DATA_BLOCK "MEStoPLC"
{ S7_Optimized_Access := 'FALSE' }
VERSION : 0.1
NON_RETAIN
   STRUCT 
      "MES.Load_Station1PartOK" : Bool;
      "MES.Load_Station1PartNG" : Bool;
      "MES.Load_Station1ReqMesDone" : Bool;
      Spare_1 : Bool;
      "MES.Load_Station2PartOK" : Bool;
      "MES.Load_Station2PartNG" : Bool;
      "MES.Load_Station2ReqMesDone" : Bool;
      Spare_2 : Bool;
      "MES.Load_Station3PartOK" : Bool;
      "MES.Load_Station3PartNG" : Bool;
      "MES.Load_Station3ReqMesDone" : Bool;
      Spare_3 : Bool;
      "MES.Load_Station4PartOK" : Bool;
      "MES.Load_Station4PartNG" : Bool;
      "MES.Load_Station4ReqMesDone" : Bool;
      Spare_4 : Bool;
      "MES.Load_Station5PartOK" : Bool;
      "MES.Load_Station5PartNG" : Bool;
      "MES.Load_Station5ReqMesDone" : Bool;
      Spare_5 : Bool;
      "MES.Load_Station6PartOK" : Bool;
      "MES.Load_Station6PartNG" : Bool;
      "MES.Load_Station6ReqMesDone" : Bool;
      Spare_6 : Bool;
      "MES.Load_Station7PartOK" : Bool;
      "MES.Load_Station7PartNG" : Bool;
      "MES.Load_Station7ReqMesDone" : Bool;
      Spare_7 : Bool;
      "MES.Load_Station8PartOK" : Bool;
      "MES.Load_Station8PartNG" : Bool;
      "MES.Load_Station8ReqMesDone" : Bool;
      Spare_8 : Bool;
      Spare_9 : Bool;
      Static_3 : Bool;
      "MES.Load_SubPart1OK" : Bool;
      "MES.Load_SubPart1tNG" : Bool;
      "MES.Load_SubPart1ReqMesDone" : Bool;
      Spare_10 : Bool;
      "MES.Load_SubPart2OK" : Bool;
      "MES.Load_SubPart2tNG" : Bool;
      "MES.Load_SubPart2ReqMesDone" : Bool;
      Spare_11 : Bool;
      "MES.Load_SubPart3OK" : Bool;
      "MES.Load_SubPart3tNG" : Bool;
      "MES.Load_SubPart3ReqMesDone" : Bool;
      Spare_12 : Bool;
      "MES.Load_SubPart4OK" : Bool;
      "MES.Load_SubPart4tNG" : Bool;
      "MES.Load_SubPart4ReqMesDone" : Bool;
      Spare_13 : Bool;
      "MES.Load_SubPart5OK" : Bool;
      "MES.Load_SubPart5tNG" : Bool;
      "MES.Load_SubPart5ReqMesDone" : Bool;
      Spare_14 : Bool;
      "MES.Load_SubPart6OK" : Bool;
      "MES.Load_SubPart6tNG" : Bool;
      "MES.Load_SubPart6ReqMesDone" : Bool;
      Spare_15 : Bool;
      "MES.Load_SubPart7OK" : Bool;
      "MES.Load_SubPart7tNG" : Bool;
      "MES.Load_SubPart7ReqMesDone" : Bool;
      Spare_16 : Bool;
      "MES.Load_SubPart8OK" : Bool;
      "MES.Load_SubPart8tNG" : Bool;
      "MES.Load_SubPart8ReqMesDone" : Bool;
      Spare : Bool;
      Spare_17 : Bool;
      "MES.Load_ResultsStored1OK" : Bool;
      "MES.Load_ResultsStored1NG" : Bool;
      "MES.Load_ResultsStored1ReqMesDone" : Bool;
      Spare_18 : Bool;
      "MES.Load_ResultsStored2OK" : Bool;
      "MES.Load_ResultsStored2NG" : Bool;
      "MES.Load_ResultsStored2ReqMesDone" : Bool;
      Spare_19 : Bool;
      "MES.Load_ResultsStored3OK" : Bool;
      "MES.Load_ResultsStored3NG" : Bool;
      "MES.Load_ResultsStored3ReqMesDone" : Bool;
      Spare_20 : Bool;
      "MES.Load_ResultsStored4OK" : Bool;
      "MES.Load_ResultsStored4NG" : Bool;
      "MES.Load_ResultsStored4ReqMesDone" : Bool;
      Spare_21 : Bool;
      "MES.Load_ResultsStored5OK" : Bool;
      "MES.Load_ResultsStored5NG" : Bool;
      "MES.Load_ResultsStored5ReqMesDone" : Bool;
      Spare_22 : Bool;
      "MES.Load_ResultsStored6OK" : Bool;
      "MES.Load_ResultsStored6NG" : Bool;
      "MES.Load_ResultsStored6ReqMesDone" : Bool;
      Spare_23 : Bool;
      "MES.Load_ResultsStored7OK" : Bool;
      "MES.Load_ResultsStored7NG" : Bool;
      "MES.Load_ResultsStored7ReqMesDone" : Bool;
      Spare_24 : Bool;
      "MES.Load_ResultsStored8OK" : Bool;
      "MES.Load_ResultsStored8NG" : Bool;
      "MES.Load_ResultsStored8ReqMesDone" : Bool;
      "MES.Load_StoveCheckInOk" : Bool;
      Static_1 : Bool;
      Spare_26 : Bool;
      Spare_27 : Bool;
      Spare_28 : Bool;
      Spare_29 : Bool;
      Spare_30 : Bool;
      Spare_31 : Bool;
      Spare_32 : Bool;
      Spare_33 : Bool;
      "MES.Unload_ResultsStored1OK" : Bool;
      "MES.Unload_ResultsStored1NG" : Bool;
      "MES.Unload_ResultsStored1ReqMesDone" : Bool;
      Spare_34 : Bool;
      "MES.Unload_ResultsStored2OK" : Bool;
      "MES.Unload_ResultsStored2NG" : Bool;
      "MES.Unload_ResultsStored2ReqMesDone" : Bool;
      Spare_35 : Bool;
      "MES.Unload_ResultsStored3OK" : Bool;
      "MES.Unload_ResultsStored3NG" : Bool;
      "MES.Unload_ResultsStored3ReqMesDone" : Bool;
      Spare_36 : Bool;
      "MES.Unload_ResultsStored4OK" : Bool;
      "MES.Unload_ResultsStored4NG" : Bool;
      "MES.Unload_ResultsStored4ReqMesDone" : Bool;
      Spare_37 : Bool;
      "MES.Unload_ResultsStored5OK" : Bool;
      "MES.Unload_ResultsStored5NG" : Bool;
      "MES.Unload_ResultsStored5ReqMesDone" : Bool;
      Spare_38 : Bool;
      "MES.Unload_ResultsStored6OK" : Bool;
      "MES.Unload_ResultsStored6NG" : Bool;
      "MES.Unload_ResultsStored6ReqMesDone" : Bool;
      Spare_39 : Bool;
      "MES.Unload_ResultsStored7OK" : Bool;
      "MES.Unload_ResultsStored7NG" : Bool;
      "MES.Unload_ResultsStored7ReqMesDone" : Bool;
      Spare_40 : Bool;
      "MES.Unload_ResultsStored8OK" : Bool;
      "MES.Unload_ResultsStored8NG" : Bool;
      "MES.Unload_ResultsStored8ReqMesDone" : Bool;
      Spare_41 : Bool;
      "MES.HeartbeatSignal" : Bool;
   END_STRUCT;


BEGIN

END_DATA_BLOCK

DATA_BLOCK "Scanner1LoadData"
{ S7_Optimized_Access := 'FALSE' }
VERSION : 0.1
NON_RETAIN
   STRUCT 
      "PLC.Station1DMXCode" : Int;
      "PLC.Station1RecipeNo" : Int;
      "PLC.PartTypeID" : String[128];
      Spare : Byte;
      "MES.ErrorCode" : Int;
      "MES.StatusBits" : DInt;
      "MES.Cycle_ID" : DInt;
      "MES.Unit_ParttypeID" : Int;
   END_STRUCT;


BEGIN

END_DATA_BLOCK

DATA_BLOCK "Station1UnLoadData"
{ S7_Optimized_Access := 'FALSE' }
VERSION : 0.1
NON_RETAIN
   STRUCT 
      "PLC.PartTypeID" : Int;
      "PLC.Station1DMXCode" : String[128];
      "PLC.Station1RecipeNo" : Int;
      "PLC.PartStatus" : Int;
      "PLC.SubPartSN1" : String[128];
      "PLC.TransferTime" : String[128];
      Spare : Byte;
      Spare_1 : Byte;
      Spare_2 : Byte;
      Spare_3 : Byte;
      Spare_4 : Byte;
      Spare_5 : Byte;
      Spare_6 : Byte;
      Spare_7 : Byte;
      Spare_8 : Byte;
      Spare_9 : Byte;
      Spare_10 : Byte;
      "MES.ErrorCode" : Int;
      "MES.ErrorMsg" : String[128];
   END_STRUCT;


BEGIN

END_DATA_BLOCK

DATA_BLOCK "Station2LoadData"
{ S7_Optimized_Access := 'FALSE' }
VERSION : 0.1
NON_RETAIN
   STRUCT 
      "PLC.PartTypeID" : Int;
      "PLC.Station2RecipeNo" : Int;
      "PLC.Station2DMXCode" : String[128];
      "PLC.SubPartSN1" : String[128];
      "MES.ErrorCode" : Int;
      "MES.StatusBits" : DInt;
      "MES.Cycle_ID" : DInt;
      "MES.Unit_ParttypeID" : Int;
   END_STRUCT;


BEGIN

END_DATA_BLOCK

DATA_BLOCK "Station2UnLoadData"
{ S7_Optimized_Access := 'FALSE' }
VERSION : 0.1
NON_RETAIN
   STRUCT 
      "PLC.PartTypeID" : Int;
      "PLC.Station2DMXCode" : String[128];
      "PLC.Station2RecipeNo" : Int;
      "PLC.PartStatus" : Int;
      "PLC.SubPartSN1" : String[128];
      "PLC.TransferTime" : String[128];
      Spare : Byte;
      Spare_1 : Byte;
      Spare_2 : Byte;
      Spare_3 : Byte;
      Spare_4 : Byte;
      Spare_5 : Byte;
      Spare_6 : Byte;
      Spare_7 : Byte;
      Spare_8 : Byte;
      Spare_9 : Byte;
      Spare_10 : Byte;
      "MES.ErrorCode" : Int;
      "MES.ErrorMsg" : String[128];
   END_STRUCT;


BEGIN

END_DATA_BLOCK

DATA_BLOCK "Station3LoadData"
{ S7_Optimized_Access := 'FALSE' }
VERSION : 0.1
NON_RETAIN
   STRUCT 
      "PLC.PartTypeID" : Int;
      "PLC.Station3RecipeNo" : Int;
      "PLC.Station3DMXCode" : String[128];
      "PLC.SubPartSN1" : String[128];
      "MES.ErrorCode" : Int;
      "MES.StatusBits" : DInt;
      "MES.Cycle_ID" : DInt;
      "MES.Unit_ParttypeID" : Int;
   END_STRUCT;


BEGIN

END_DATA_BLOCK

DATA_BLOCK "Station4LoadData"
{ S7_Optimized_Access := 'FALSE' }
VERSION : 0.1
NON_RETAIN
   STRUCT 
      "PLC.PartTypeID" : Int;
      "PLC.Station4RecipeNo" : Int;
      "PLC.Station4DMXCode" : String[128];
      "PLC.SubPartSN1" : String[128];
      "MES.ErrorCode" : Int;
      "MES.StatusBits" : DInt;
      "MES.Cycle_ID" : DInt;
      "MES.Unit_ParttypeID" : Int;
   END_STRUCT;


BEGIN

END_DATA_BLOCK

DATA_BLOCK "Station4UnLoadData"
{ S7_Optimized_Access := 'FALSE' }
VERSION : 0.1
NON_RETAIN
   STRUCT 
      "PLC.PartTypeID" : Int;
      "PLC.Station4DMXCode" : String[50];
      "PLC.Station4RecipeNo" : Int;
      "PLC.PartStatus" : Int;
      "PLC.SubPartSN1" : String[50];
      "PLC.TransferTime" : String[50];
      Spare : Byte;
      Spare_1 : Byte;
      Spare_2 : Byte;
      Spare_3 : Byte;
      Spare_4 : Byte;
      Spare_5 : Byte;
      Spare_6 : Byte;
      Spare_7 : Byte;
      Spare_8 : Byte;
      Spare_9 : Byte;
      Spare_10 : Byte;
      "MES.ErrorCode" : Int;
      "MES.ErrorMsg" : String[60];
   END_STRUCT;


BEGIN

END_DATA_BLOCK

DATA_BLOCK "Station5LoadData"
{ S7_Optimized_Access := 'FALSE' }
VERSION : 0.1
NON_RETAIN
   STRUCT 
      "PLC.PartTypeID" : Int;
      "PLC.Station5RecipeNo" : Int;
      "PLC.Station5DMXCode" : String[128];
      "PLC.SubPartSN1" : String[128];
      "MES.ErrorCode" : Int;
      "MES.StatusBits" : DInt;
      "MES.Cycle_ID" : DInt;
      "MES.Unit_ParttypeID" : Int;
   END_STRUCT;


BEGIN

END_DATA_BLOCK

DATA_BLOCK "Station5UnLoadData"
{ S7_Optimized_Access := 'FALSE' }
VERSION : 0.1
NON_RETAIN
   STRUCT 
      "PLC.PartTypeID" : Int;
      "PLC.Station5DMXCode" : String[50];
      "PLC.Station5RecipeNo" : Int;
      "PLC.PartStatus" : Int;
      "PLC.SubPartSN1" : String[50];
      "PLC.TransferTime" : String[50];
      "PLC.ShaftGlueIVPro" : Int;
      "PLC.ShaftGlueResult" : Int;
      "PLC.ShaftGlueIVScore1" : Int;
      "PLC.ShaftGlueIVScore2" : Int;
      "PLC.ShaftGlueIVScore3" : Int;
      "PLC.ShaftGlueIVScore4" : Int;
      "PLC.ShaftMagnetIVPro" : Int;
      "PLC.MagnetGlueResult" : Int;
      "PLC.MagnetIVScore" : Int;
      "PLC.GluePro" : Int;
      "PLC.NGCode" : Int;
      Spare_5 : Int;
      Spare_6 : Int;
      Spare_7 : Int;
      Spare_8 : Int;
      Spare_9 : Int;
      Spare_10 : Int;
      "MES.ErrorCode" : Int;
      "MES.ErrorMsg" : String[60];
   END_STRUCT;


BEGIN

END_DATA_BLOCK

DATA_BLOCK "Station6LoadData"
{ S7_Optimized_Access := 'FALSE' }
VERSION : 0.1
NON_RETAIN
   STRUCT 
      "PLC.PartTypeID" : Int;
      "PLC.Station6RecipeNo" : Int;
      "PLC.Station6DMXCode" : String[128];
      "PLC.SubPartSN1" : String[128];
      "MES.ErrorCode" : Int;
      "MES.StatusBits" : DInt;
      "MES.Cycle_ID" : DInt;
      "MES.Unit_ParttypeID" : Int;
   END_STRUCT;


BEGIN

END_DATA_BLOCK

DATA_BLOCK "Station6UnLoadData"
{ S7_Optimized_Access := 'FALSE' }
VERSION : 0.1
NON_RETAIN
   STRUCT 
      "PLC.PartTypeID" : Int;
      "PLC.Station6DMXCode" : String[50];
      "PLC.Station6RecipeNo" : Int;
      "PLC.PartStatus" : Int;
      "PLC.SubPartSN1" : String[50];
      "PLC.TransferTime" : String[50];
      Spare : Byte;
      Spare_1 : Byte;
      Spare_2 : Byte;
      Spare_3 : Byte;
      Spare_4 : Byte;
      Spare_5 : Byte;
      Spare_6 : Byte;
      Spare_7 : Byte;
      Spare_8 : Byte;
      Spare_9 : Byte;
      Spare_10 : Byte;
      "MES.ErrorCode" : Int;
      "MES.ErrorMsg" : String[60];
   END_STRUCT;


BEGIN

END_DATA_BLOCK

DATA_BLOCK "Station7UnLoadData"
{ S7_Optimized_Access := 'FALSE' }
VERSION : 0.1
NON_RETAIN
   STRUCT 
      "PLC.PartTypeID" : Int;
      "PLC.Station7DMXCode" : String[50];
      "PLC.Station7RecipeNo" : Int;
      "PLC.PartStatus" : Int;
      "PLC.SubPartSN1" : String[50];
      "PLC.TransferTime" : String[50];
      "PLC.Power" : Real;
      "PLC.Displacement" : Real;
      "PLC.Program" : Int;
      "PLC.NGCode" : Int;
      Spare_2 : Byte;
      Spare_3 : Byte;
      Spare_4 : Byte;
      Spare_5 : Byte;
      Spare_6 : Byte;
      Spare_7 : Byte;
      Spare_8 : Byte;
      "MES.ErrorCode" : Int;
      "MES.ErrorMsg" : String[60];
   END_STRUCT;


BEGIN

END_DATA_BLOCK

DATA_BLOCK "Station8UnLoadData"
{ S7_Optimized_Access := 'FALSE' }
VERSION : 0.1
NON_RETAIN
   STRUCT 
      "PLC.PartTypeID" : Int;
      "PLC.Station7DMXCode" : String[50];
      "PLC.Station7RecipeNo" : Int;
      "PLC.PartStatus" : Int;
      "PLC.SubPartSN1" : String[50];
      "PLC.TransferTime" : String[50];
      "PLC.Power" : Real;
      "PLC.Displacement" : Real;
      Spare : Byte;
      Spare_1 : Byte;
      Spare_2 : Byte;
      Spare_3 : Byte;
      Spare_4 : Byte;
      Spare_5 : Byte;
      Spare_6 : Byte;
      Spare_7 : Byte;
      Spare_8 : Byte;
      "MES.ErrorCode" : Int;
      "MES.ErrorMsg" : String[60];
   END_STRUCT;


BEGIN

END_DATA_BLOCK

DATA_BLOCK "PartDataManage_Part1_DB"
{ S7_Optimized_Access := 'TRUE' }
VERSION : 0.1
NON_RETAIN
"PartDataManage"

BEGIN

END_DATA_BLOCK

DATA_BLOCK "PartDataManage_Part4_DB"
{ S7_Optimized_Access := 'TRUE' }
VERSION : 0.1
NON_RETAIN
"PartDataManage"

BEGIN

END_DATA_BLOCK

DATA_BLOCK "ST10_SystemModeFB_iDB"
{ S7_Optimized_Access := 'TRUE' }
VERSION : 0.1
NON_RETAIN
"SystemMode"

BEGIN

END_DATA_BLOCK

DATA_BLOCK "ChangeOver_DB"
{ S7_Optimized_Access := 'FALSE' }
VERSION : 0.1
   STRUCT 
      Robot_1 : Struct
         Req_RobotToMaintenancePos : Bool;
         Req_RobotToHomePos : Bool;
         Sensor_3 : Bool;
         Sensor_4 : Bool;
         Sensor_5 : Bool;
         Sensor_6 : Bool;
         Sensor_7 : Bool;
         Sensor_8 : Bool;
         EmptyProcess : Bool;
         EmptyFinish : Bool;
         Spare : Bool;
         HMI_MaintenancePosReqSel : Bool;
         HMI_MaintenancePosActive : Bool;
         MaintenancePosReqSelFlag : Bool;
         HMI_MaintenanceHomeReq : Bool;
         NoTaskRunning : Bool;
         Spare_6 : Bool;
         Step : Int;
      END_STRUCT;
      Robot_2 : Struct
         Req_RobotToMaintenancePos : Bool;
         Req_RobotToHomePos : Bool;
         Sensor_3 : Bool;
         Sensor_4 : Bool;
         Sensor_5 : Bool;
         Sensor_6 : Bool;
         Sensor_7 : Bool;
         Sensor_8 : Bool;
         EmptyProcess : Bool;
         EmptyFinish : Bool;
         Spare : Bool;
         HMI_MaintenancePosReqSel : Bool;
         HMI_MaintenancePosActive : Bool;
         MaintenancePosReqSelFlag : Bool;
         HMI_MaintenanceHomeReq : Bool;
         NoTaskRunning : Bool;
         Spare_6 : Bool;
         Step : Int;
      END_STRUCT;
      Robot_3 : Struct
         Req_RobotToMaintenancePos : Bool;
         Req_RobotToHomePos : Bool;
         Sensor_3 : Bool;
         Sensor_4 : Bool;
         Sensor_5 : Bool;
         Sensor_6 : Bool;
         Sensor_7 : Bool;
         Sensor_8 : Bool;
         EmptyProcess : Bool;
         EmptyFinish : Bool;
         Spare : Bool;
         HMI_MaintenancePosReqSel : Bool;
         HMI_MaintenancePosActive : Bool;
         MaintenancePosReqSelFlag : Bool;
         HMI_MaintenanceHomeReq : Bool;
         NoTaskRunning : Bool;
         Spare_6 : Bool;
         Step : Int;
      END_STRUCT;
      H_Line : Struct
         Sensor_1 : Bool;
         Sensor_2 : Bool;
         Sensor_3 : Bool;
         Sensor_4 : Bool;
         Sensor_5 : Bool;
         Sensor_6 : Bool;
         Sensor_7 : Bool;
         Sensor_8 : Bool;
         Sensor_9 : Bool;
         Sensor_10 : Bool;
         Sensor_11 : Bool;
         Sensor_12 : Bool;
         Sensor_13 : Bool;
         Sensor_14 : Bool;
         Sensor_15 : Bool;
         Sensor_16 : Bool;
         EmptyProcess : Bool;
         EmptyFinish : Bool;
         Spare : Bool;
         Spare_1 : Bool;
         Spare_2 : Bool;
         Spare_3 : Bool;
         Spare_4 : Bool;
         Spare_5 : Bool;
         Spare_6 : Bool;
         Step : Int;
      END_STRUCT;
      J_Line : Struct
         Sensor_1 : Bool;
         Sensor_2 : Bool;
         Sensor_3 : Bool;
         Sensor_4 : Bool;
         Sensor_5 : Bool;
         Sensor_6 : Bool;
         Sensor_7 : Bool;
         Sensor_8 : Bool;
         Sensor_9 : Bool;
         Sensor_10 : Bool;
         Sensor_11 : Bool;
         Sensor_12 : Bool;
         Sensor_13 : Bool;
         Sensor_14 : Bool;
         Sensor_15 : Bool;
         Sensor_16 : Bool;
         EmptyProcess : Bool;
         EmptyFinish : Bool;
         Spare : Bool;
         Spare_1 : Bool;
         Spare_2 : Bool;
         Spare_3 : Bool;
         Spare_4 : Bool;
         Spare_5 : Bool;
         Spare_6 : Bool;
         Step : Int;
      END_STRUCT;
      K_Line : Struct
         Sensor_1 : Bool;
         Sensor_2 : Bool;
         Sensor_3 : Bool;
         Sensor_4 : Bool;
         Sensor_5 : Bool;
         Sensor_6 : Bool;
         Sensor_7 : Bool;
         Sensor_8 : Bool;
         Sensor_9 : Bool;
         Sensor_10 : Bool;
         Sensor_11 : Bool;
         Sensor_12 : Bool;
         Sensor_13 : Bool;
         Sensor_14 : Bool;
         Sensor_15 : Bool;
         Sensor_16 : Bool;
         EmptyProcess : Bool;
         EmptyFinish : Bool;
         Spare : Bool;
         Spare_1 : Bool;
         Spare_2 : Bool;
         Spare_3 : Bool;
         Spare_4 : Bool;
         Spare_5 : Bool;
         Spare_6 : Bool;
         Step : Int;
      END_STRUCT;
      L_Line : Struct
         Sensor_1 : Bool;
         Sensor_2 : Bool;
         Sensor_3 : Bool;
         Sensor_4 : Bool;
         Sensor_5 : Bool;
         Sensor_6 : Bool;
         Sensor_7 : Bool;
         Sensor_8 : Bool;
         Sensor_9 : Bool;
         Sensor_10 : Bool;
         Sensor_11 : Bool;
         Sensor_12 : Bool;
         Sensor_13 : Bool;
         Sensor_14 : Bool;
         Sensor_15 : Bool;
         Sensor_16 : Bool;
         EmptyProcess : Bool;
         EmptyFinish : Bool;
         Spare : Bool;
         Spare_1 : Bool;
         Spare_2 : Bool;
         Spare_3 : Bool;
         Spare_4 : Bool;
         Spare_5 : Bool;
         Spare_6 : Bool;
         Step : Int;
      END_STRUCT;
      Global : Struct
         AllFixtureScanCompareOk : Bool;
         ChangeOverRequest : Bool;
         ChangeOverToolScanFlag : Bool;
         ManualModeFlag : Bool;
         ScanFixtureFlag : Bool;
         Station_empty : Bool;
         ChangeOverSelected : Bool;
         ScanFixtureFlag_ChangeOver : Bool;
         A1_TableScanStart : Bool;
         A2_TableScanStart : Bool;
         Hmi_Confirm_ChangeOver : Bool;
         ChangeOverActive : Bool;
         Hmi_ForceChangeOver : Bool;
         Spare_13 : Bool;
         Spare_14 : Bool;
         Spare_15 : Bool;
      END_STRUCT;
      P : Array[0..20] of Bool;
      "Time" {InstructionName := 'TOF_TIME'; LibVersion := '1.0'; S7_SetPoint := 'False'} : Array[0..3] of TOF_TIME;
      Robot1 : Struct
         Ring1Weight : Int;
         ShaftWeight : Int;
         MagnetWeight : Int;
         Ring2Weight : Int;
      END_STRUCT;
      Robot2 : Struct
         Ring1Weight : Int;
         ShaftWeight : Int;
         MagnetWeight : Int;
         Ring2Weight : Int;
      END_STRUCT;
      Robot3 : Struct
         Ring1Weight : Int;
         ShaftWeight : Int;
         MagnetWeight : Int;
         Ring2Weight : Int;
      END_STRUCT;
   END_STRUCT;


BEGIN

END_DATA_BLOCK

DATA_BLOCK "AutoProcessDataPopUp_DB"
{ S7_Optimized_Access := 'TRUE' }
VERSION : 0.1
NON_RETAIN
"AutoProcessDataPopUp"

BEGIN

END_DATA_BLOCK

DATA_BLOCK "AutoProcess_HMI"
{ S7_Optimized_Access := 'TRUE' }
VERSION : 0.1
NON_RETAIN
   VAR 
      IndexProcess : Int;   // 1 A_ScanRotate, 2 F_Robot1Grip1, 3 F_Robot1Grip2, 4 B_Press1, 5 C_Glue, 6 F_Robot2Grip1, 7 F_Robot2Grip2, 8 C_GlueNGBuffer, 9 C_MagnScanNGBuffer, 10 B_Press2, 11 F_Robot3Grip1, 12 F_Robot3Grip2, 13 H_ShafeLine, 14 J_ShafeLine, 15 K_ShafeLine, 16 L_ShafeLine
      ActualSHowingData { S7_SetPoint := 'False'} : "ProcessData";
      Data_handling : Struct
         DeleteData : Bool;
         UpdateData_switch : Bool;
         UpdateData_Confirm : Bool;   // 1. step - request to confirm old new data
         FinalConfirm_Write : Bool;   // 2.  final acceptance for data update
         ChangePending : Bool;   // changes are ready for actual index
         ConfirmDialogActive : Bool;   // Confirm dialog active
         LastIndex : Int;   // internal - memory for last index
      END_STRUCT;
      StationHasProduct : Array[1..16] of Bool;
   END_VAR


BEGIN

END_DATA_BLOCK

DATA_BLOCK "ST10_Flow11_A2TableScan_iDB"
{ S7_Optimized_Access := 'TRUE' }
VERSION : 0.1
NON_RETAIN
"ST10_Flow11_A2TableScan"

BEGIN

END_DATA_BLOCK

DATA_BLOCK "ST10_Flow21_HShaftLifting_iDB"
{ S7_Optimized_Access := 'TRUE' }
VERSION : 0.1
NON_RETAIN
"ST10_Flow21_HShaftLifting"

BEGIN

END_DATA_BLOCK

DATA_BLOCK "ST10_Flow23_KReserveLifting_iDB"
{ S7_Optimized_Access := 'TRUE' }
VERSION : 0.1
NON_RETAIN
"ST10_Flow23_KReserveLifting"

BEGIN

END_DATA_BLOCK

DATA_BLOCK "ST10_Flow24_LUnloadingTrans_iDB"
{ S7_Optimized_Access := 'TRUE' }
VERSION : 0.1
NON_RETAIN
"ST10_Flow24_LUnloadingTrans"

BEGIN

END_DATA_BLOCK

DATA_BLOCK "ST10_Flow27_KReserveLoad&Unload_iDB"
{ S7_Optimized_Access := 'TRUE' }
VERSION : 0.1
NON_RETAIN
"ST10_Flow27_KReserveLoad&Unload"

BEGIN

END_DATA_BLOCK

DATA_BLOCK "ST10_Flow8_FRobot_2_iDB"
{ S7_Optimized_Access := 'TRUE' }
VERSION : 0.1
NON_RETAIN
"ST10_Flow8_FRobot_2"

BEGIN

END_DATA_BLOCK

DATA_BLOCK "ST10_MaterialGate2_DB"
{ S7_Optimized_Access := 'FALSE' }
VERSION : 0.1
NON_RETAIN
"SafetyGate"

BEGIN

END_DATA_BLOCK

DATA_BLOCK "ST10_MaterialGate4_DB"
{ S7_Optimized_Access := 'FALSE' }
VERSION : 0.1
NON_RETAIN
"SafetyGate"

BEGIN

END_DATA_BLOCK

DATA_BLOCK "ST10_MaterialGate5_DB"
{ S7_Optimized_Access := 'FALSE' }
VERSION : 0.1
NON_RETAIN
"SafetyGate"

BEGIN

END_DATA_BLOCK

DATA_BLOCK "ST10_MaterialGate6_DB"
{ S7_Optimized_Access := 'FALSE' }
VERSION : 0.1
NON_RETAIN
"SafetyGate"

BEGIN

END_DATA_BLOCK

DATA_BLOCK "ST10_NGGate2_DB"
{ S7_Optimized_Access := 'FALSE' }
VERSION : 0.1
NON_RETAIN
"SafetyGate"

BEGIN

END_DATA_BLOCK

DATA_BLOCK "ST10_SafetyGate1_DB"
{ S7_Optimized_Access := 'FALSE' }
VERSION : 0.1
NON_RETAIN
"SafetyGate"

BEGIN

END_DATA_BLOCK

DATA_BLOCK "ST10_SafetyGate2_DB"
{ S7_Optimized_Access := 'FALSE' }
VERSION : 0.1
NON_RETAIN
"SafetyGate"

BEGIN

END_DATA_BLOCK

DATA_BLOCK "ST10_SafetyGate3_DB"
{ S7_Optimized_Access := 'FALSE' }
VERSION : 0.1
NON_RETAIN
"SafetyGate"

BEGIN

END_DATA_BLOCK

DATA_BLOCK "ST10_SafetyGate4_DB"
{ S7_Optimized_Access := 'FALSE' }
VERSION : 0.1
NON_RETAIN
"SafetyGate"

BEGIN

END_DATA_BLOCK

DATA_BLOCK "ST10_SafetyGate5_DB"
{ S7_Optimized_Access := 'FALSE' }
VERSION : 0.1
NON_RETAIN
"SafetyGate"

BEGIN

END_DATA_BLOCK

DATA_BLOCK "ST10_SafetyGate8_DB"
{ S7_Optimized_Access := 'FALSE' }
VERSION : 0.1
NON_RETAIN
"SafetyGate"

BEGIN

END_DATA_BLOCK

DATA_BLOCK "ST10_SafetyGate9_DB"
{ S7_Optimized_Access := 'FALSE' }
VERSION : 0.1
NON_RETAIN
"SafetyGate"

BEGIN

END_DATA_BLOCK

DATA_BLOCK "ST10_SafetyGate_InterfaceDB"
{ S7_Optimized_Access := 'TRUE' }
VERSION : 0.1
NON_RETAIN
   VAR 
      aDev : Array[1..20] of "SafetyGateUDT";
      SafetyDoorLamp { S7_SetPoint := 'True'} : Array[1..20] of Bool;
      H : Struct
         Status_1 : Int;
         Status_2 : Int;
         Status_3 : Int;
         p : Array[0..20] of Bool;
      END_STRUCT;
      J : Struct
         Status_1 : Int;
         Status_2 : Int;
         Status_3 : Int;
         p : Array[0..20] of Bool;
      END_STRUCT;
      K : Struct
         Status_1 : Int;
         Status_2 : Int;
         Status_3 : Int;
         p : Array[0..20] of Bool;
      END_STRUCT;
      L : Struct
         Status_1 : Int;
         Status_2 : Int;
         Status_3 : Int;
         p : Array[0..20] of Bool;
      END_STRUCT;
   END_VAR


BEGIN

END_DATA_BLOCK

DATA_BLOCK "ST10_Stopper_FB_DB"
{ S7_Optimized_Access := 'TRUE' }
VERSION : 0.1
NON_RETAIN
"ST10_Stopper_FB"

BEGIN

END_DATA_BLOCK

DATA_BLOCK "ST10_Stopper_InterfaceDB"
{ S7_Optimized_Access := 'TRUE' }
VERSION : 0.1
NON_RETAIN
   VAR 
      aDev : Array[1..5] of "ST_Stopper";
      Command : Array[1..5] of "UDT_Stopper_FB";
   END_VAR


BEGIN

END_DATA_BLOCK

DATA_BLOCK "ST10_PLC_PutDB"
{ S7_Optimized_Access := 'FALSE' }
VERSION : 0.1
NON_RETAIN
   STRUCT 
      OutData : Struct
         Global : Struct
            Beat : Bool;
            AutoRunning : Bool;
            Alarm : Bool;
            Spare_1 : Bool;
            Spare_2 : Bool;
            Spare_3 : Bool;
            Spare_4 : Bool;
            Spare_5 : Bool;
            Spare_6 : Bool;
            Spare_7 : Bool;
            Spare_8 : Bool;
            Spare_9 : Bool;
            Spare_10 : Bool;
            Spare_11 : Bool;
            Spare_12 : Bool;
            Spare_13 : Bool;
         END_STRUCT;
         Control : Struct
            PalletOut : Bool;
            Spare_16 : Bool;
            Spare_1 : Bool;
            Spare_2 : Bool;
            Spare_3 : Bool;
            Spare_4 : Bool;
            Spare_5 : Bool;
            Spare_6 : Bool;
            Spare_7 : Bool;
            Spare_8 : Bool;
            Spare_9 : Bool;
            Spare_10 : Bool;
            Spare_11 : Bool;
            Spare_12 : Bool;
            Spare_13 : Bool;
            Spare_14 : Byte;
            Spare_15 : Byte;
         END_STRUCT;
         Data : Struct
            Spare_5 : Int;
            Spare_4 : Int;
            Spare_1 : Int;
            Spare_2 : Int;
            Spare_6 : Int;   // Min
            Spare_3 : Array[0..83] of Byte;
         END_STRUCT;
      END_STRUCT;
   END_STRUCT;


BEGIN

END_DATA_BLOCK

DATA_BLOCK "KeyenceSR1000Ctrl_801A1DB"
{ S7_Optimized_Access := 'FALSE' }
VERSION : 0.1
NON_RETAIN
"KeyenceSR1000Ctrl"

BEGIN

END_DATA_BLOCK

DATA_BLOCK "KeyenceSR1000Ctrl_803A1DB"
{ S7_Optimized_Access := 'FALSE' }
VERSION : 0.1
NON_RETAIN
"KeyenceSR1000Ctrl"

BEGIN

END_DATA_BLOCK

DATA_BLOCK "KeyenceSR1000Ctrl_805A1DB"
{ S7_Optimized_Access := 'FALSE' }
VERSION : 0.1
NON_RETAIN
"KeyenceSR1000Ctrl"

BEGIN

END_DATA_BLOCK

DATA_BLOCK "KeyenceSR1000Ctrl_806A1DB"
{ S7_Optimized_Access := 'FALSE' }
VERSION : 0.1
NON_RETAIN
"KeyenceSR1000Ctrl"

BEGIN

END_DATA_BLOCK

DATA_BLOCK "KeyenceSR1000Ctrl_807A1DB"
{ S7_Optimized_Access := 'FALSE' }
VERSION : 0.1
NON_RETAIN
"KeyenceSR1000Ctrl"

BEGIN

END_DATA_BLOCK

DATA_BLOCK "IAI_A1"
{ S7_Optimized_Access := 'FALSE' }
VERSION : 0.1
   STRUCT 
      In : Struct
         iInterlock : Bool;
         "iManJog+" : Bool;
         "iManJog-" : Bool;
         iAutoStart : Bool;
         iHome : Bool;
         iCancelTask : Bool;
         iPauseTask : Bool;
         iManStart : Bool;
         iManListStart : Bool;
         iLimitSwitchActive : Bool;
         iLimitSoftActive : Bool;
         iRunningTimeout : Time;
         iHomingTimeout : Time;
         iAutoPosition : DInt;
         iAutoVelocity : Int;
         iManListPosition : DInt;
         iManListVelocity : Int;
         iManListNumber : Int;
         iManPosition : DInt;
         iManVelocity : Int;
         iMode : Int;
      END_STRUCT;
      Out : Struct
         oReady : Bool;
         oWarning : Bool;
         oError : Bool;
         oInterlock : Bool;
         oServoEnable : Bool;
         oRunning : Bool;
         oHoming : Bool;
         oHomeRef : Bool;
         oServoPosOK : Bool;
         oErrorCode : Int;
         oStatus : Int;
         oActPosition : DInt;
         oManualListPos : DInt;
      END_STRUCT;
      IO : Struct
         ioManEnale : Bool;
         ioAutoEnale : Bool;
      END_STRUCT;
      Spare : Struct
         S : Array[0..100] of Byte;
      END_STRUCT;
      Manual : Struct
         Index : Int;
         Pos : Array[1..20] of Struct
            Pos : Real;
            Vel : Int;
         END_STRUCT;
      END_STRUCT;
      Auto : Struct
         Index : Int;
         Pos : Array[1..20] of Struct
            Pos : Real;
            Vel : Int;
         END_STRUCT;
      END_STRUCT;
      Interlock : Struct
         Active : Bool;
         Case1 : Bool;
         Case2 : Bool;
         Case3 : Bool;
         Case4 : Bool;
         Case5 : Bool;
         Case6 : Bool;
         Case7 : Bool;
         Case8 : Bool;
         Case9 : Bool;
         Case10 : Bool;
      END_STRUCT;
      PositionOk : Array[1..20] of Bool;
      Home_Pos : Struct
         "Home Pos Pls" : Bool;
         "Arrow indication" : Int;
         "Process prompt" : Int;
         "Button prompt" : Int;
      END_STRUCT;
   END_STRUCT;


BEGIN
   In.iLimitSwitchActive := true;
   In.iLimitSoftActive := true;
   Manual.Index := 1;
   Auto.Index := 1;

END_DATA_BLOCK

DATA_BLOCK "IAI_A3"
{ S7_Optimized_Access := 'FALSE' }
VERSION : 0.1
NON_RETAIN
   STRUCT 
      In : Struct
         iInterlock : Bool;
         "iManJog+" : Bool;
         "iManJog-" : Bool;
         iAutoStart : Bool;
         iHome : Bool;
         iCancelTask : Bool;
         iPauseTask : Bool;
         iManStart : Bool;
         iManListStart : Bool;
         iLimitSwitchActive : Bool;
         iLimitSoftActive : Bool;
         iRunningTimeout : Time;
         iHomingTimeout : Time;
         iAutoPosition : DInt;
         iAutoVelocity : Int;
         iManListPosition : DInt;
         iManListVelocity : Int;
         iManListNumber : Int;
         iManPosition : DInt;
         iManVelocity : Int;
         iMode : Int;
      END_STRUCT;
      Out : Struct
         oReady : Bool;
         oWarning : Bool;
         oError : Bool;
         oInterlock : Bool;
         oServoEnable : Bool;
         oRunning : Bool;
         oHoming : Bool;
         oHomeRef : Bool;
         oServoPosOK : Bool;
         oErrorCode : Int;
         oStatus : Int;
         oActPosition : DInt;
         oManualListPos : DInt;
      END_STRUCT;
      IO : Struct
         ioManEnale : Bool;
         ioAutoEnale : Bool;
      END_STRUCT;
      Spare : Struct
         S : Array[0..100] of Byte;
      END_STRUCT;
      Manual : Struct
         Index : Int;
         Pos : Array[1..20] of Struct
            Pos : Real;
            Vel : Int;
         END_STRUCT;
      END_STRUCT;
      Auto : Struct
         Index : Int;
         Pos : Array[1..20] of Struct
            Pos : Real;
            Vel : Int;
         END_STRUCT;
      END_STRUCT;
      Interlock : Struct
         Active : Bool;
         Case1 : Bool;
         Case2 : Bool;
         Case3 : Bool;
         Case4 : Bool;
         Case5 : Bool;
         Case6 : Bool;
         Case7 : Bool;
         Case8 : Bool;
         Case9 : Bool;
         Case10 : Bool;
      END_STRUCT;
      PositionOk : Array[1..20] of Bool;
      Home_Pos : Struct
         "Home Pos Pls" : Bool;
         "Arrow indication" : Int;
         "Process prompt" : Int;
         "Button prompt" : Int;
      END_STRUCT;
   END_STRUCT;


BEGIN
   In.iLimitSwitchActive := true;
   In.iLimitSoftActive := true;
   Manual.Index := 1;
   Auto.Index := 1;

END_DATA_BLOCK

DATA_BLOCK "ModeDB"
{ S7_Optimized_Access := 'FALSE' }
VERSION : 0.1
NON_RETAIN
   STRUCT 
      Gen : "ModeGenStruct";
   END_STRUCT;


BEGIN

END_DATA_BLOCK

DATA_BLOCK "KukaRobot1_CtrlDB"
{ S7_Optimized_Access := 'FALSE' }
VERSION : 0.1
"KukaRobot1_Ctrl"

BEGIN

END_DATA_BLOCK

DATA_BLOCK "KukaRobot2_CtrlDB"
{ S7_Optimized_Access := 'FALSE' }
VERSION : 0.1
"KukaRobot2_Ctrl"

BEGIN

END_DATA_BLOCK

DATA_BLOCK "Robot_DB"
{ S7_Optimized_Access := 'FALSE' }
VERSION : 0.1
NON_RETAIN
   STRUCT 
      LoadNG_1 : Array[1..5] of Bool;
      LoadNG_2 : Array[1..5] of Bool;
      LoadNG_3 : Array[1..5] of Bool;
      UnLoadNG_1 : Array[1..5] of Bool;
      UnLoadNG_2 : Array[1..5] of Bool;
      UnLoadNG_3 : Array[1..5] of Bool;
      P : Array[1..16] of Bool;
      RobotFlag_1 : Array[1..8] of Bool;
      RobotFlag_2 : Array[1..8] of Bool;
      RobotFlag_3 : Array[1..8] of Bool;
      RobotSpeed : Array[1..8] of USInt;
      TON {InstructionName := 'TON_TIME'; LibVersion := '1.0'; S7_SetPoint := 'False'} : Array[1..18] of TON_TIME;
      Control : Struct
         Robot1GripControl : Bool;
         Robot2GripControl : Bool;
         Robot3GripControl : Bool;
      END_STRUCT;
      Robot_1 : Struct
         PalletCount_1 : Int;
         GripCompareCodeOK_1 : Bool;
         GripCompareCodeOK_2 : Bool;
         GripCompareCodeOK_3 : Bool;
         GripCompareCodeOK_4 : Bool;
         GripCompareCodeOK : Bool;
         Spare_8 : Bool;
         Spare_6 : Bool;
         Spare_7 : Bool;
         SpeedChangeFlag : Bool;
         MasteringTest_Req : Bool;
         BrakeTest_Req : Bool;
         Spare_11 : Bool;
         Spare_12 : Bool;
         Spare_13 : Bool;
         Spare_14 : Bool;
         Spare_15 : Bool;
         SpeedCount : Int;
      END_STRUCT;
      Robot_2 : Struct
         PalletCount_1 : Int;
         PalletCount_2 : Int;
         GripCompareCodeOK_1 : Bool;
         GripCompareCodeOK_2 : Bool;
         GripCompareCodeOK_3 : Bool;
         GripCompareCodeOK_4 : Bool;
         GripCompareCodeOK : Bool;
         Spare_5 : Bool;
         Spare_6 : Bool;
         Spare_7 : Bool;
         SpeedChangeFlag : Bool;
         MasteringTest_Req : Bool;
         BrakeTest_Req : Bool;
         Spare_11 : Bool;
         Spare_12 : Bool;
         Spare_13 : Bool;
         Spare_14 : Bool;
         Spare_15 : Bool;
         SpeedCount : Int;
      END_STRUCT;
      Robot_3 : Struct
         PalletCount_1 : Int;
         PalletCount_2 : Int;
         GripCompareCodeOK_1 : Bool;
         GripCompareCodeOK_2 : Bool;
         GripCompareCodeOK_3 : Bool;
         GripCompareCodeOK_4 : Bool;
         GripCompareCodeOK : Bool;
         Spare_5 : Bool;
         Spare_6 : Bool;
         Spare_7 : Bool;
         SpeedChangeFlag : Bool;
         MasteringTest_Req : Bool;
         BrakeTest_Req : Bool;
         Spare_11 : Bool;
         Spare_12 : Bool;
         Spare_13 : Bool;
         Spare_14 : Bool;
         Spare_15 : Bool;
         SpeedCount : Int;
      END_STRUCT;
   END_STRUCT;


BEGIN

END_DATA_BLOCK

DATA_BLOCK "ServoV90_A2"
{ S7_Optimized_Access := 'FALSE' }
VERSION : 0.1
NON_RETAIN
   STRUCT 
      In : Struct
         iInterlock : Bool;
         "iManJog+" : Bool;
         "iManJog-" : Bool;
         iAutoStart : Bool;
         iHome : Bool;
         iCancelTask : Bool;
         iPauseTask : Bool;
         iManStart : Bool;
         iManListStart : Bool;
         iLimitSwitchActive : Bool;
         iLimitSoftActive : Bool;
         iRunningTimeout : Time;
         iHomingTimeout : Time;
         iAutoPosition : DInt;
         iAutoVelocity : Int;
         iManListPosition : DInt;
         iManListVelocity : Int;
         iManListNumber : Int;
         iManPosition : DInt;
         iManVelocity : Int;
         iMode : Int;
      END_STRUCT;
      Out : Struct
         oReady : Bool;
         oWarning : Bool;
         oError : Bool;
         oInterlock : Bool;
         oServoEnable : Bool;
         oRunning : Bool;
         oHoming : Bool;
         oHomeRef : Bool;
         oServoPosOK : Bool;
         oErrorCode : Int;
         oStatus : Int;
         oActPosition : DInt;
         oManualListPos : DInt;
      END_STRUCT;
      IO : Struct
         ioManEnale : Bool;
         ioAutoEnale : Bool;
      END_STRUCT;
      Spare : Struct
         S : Array[0..100] of Byte;
      END_STRUCT;
      Manual : Struct
         Index : Int;
         Pos : Array[1..20] of Struct
            Pos : DInt;
            Vel : Int;
         END_STRUCT;
      END_STRUCT;
      Auto : Struct
         Index : Int;
         Pos : Array[1..20] of Struct
            Pos : DInt;
            Vel : Int;
         END_STRUCT;
      END_STRUCT;
      Interlock : Struct
         Active : Bool;
         Case1 : Bool;
         Case2 : Bool;
         Case3 : Bool;
         Case4 : Bool;
         Case5 : Bool;
         Case6 : Bool;
         Case7 : Bool;
         Case8 : Bool;
         Case9 : Bool;
         Case10 : Bool;
      END_STRUCT;
      PositionOk : Array[1..20] of Bool;
      Home_Pos : Struct
         "Home Pos Pls" : Bool;
         "Arrow indication" : Int;
         "Process prompt" : Int;
         "Button prompt" : Int;
      END_STRUCT;
   END_STRUCT;


BEGIN
   In.iInterlock := TRUE;
   In."iManJog+" := FALSE;
   In."iManJog-" := FALSE;
   In.iAutoStart := FALSE;
   In.iHome := FALSE;
   In.iCancelTask := FALSE;
   In.iPauseTask := FALSE;
   In.iManStart := FALSE;
   In.iManListStart := FALSE;
   In.iLimitSwitchActive := TRUE;
   In.iLimitSoftActive := TRUE;
   In.iRunningTimeout := T#0MS;
   In.iHomingTimeout := T#0MS;
   In.iAutoPosition := 0;
   In.iAutoVelocity := 0;
   In.iManListPosition := 0;
   In.iManListVelocity := 0;
   In.iManListNumber := 0;
   In.iManPosition := 0;
   In.iManVelocity := 0;
   In.iMode := 0;
   Out.oReady := FALSE;
   Out.oWarning := FALSE;
   Out.oError := TRUE;
   Out.oInterlock := TRUE;
   Out.oServoEnable := FALSE;
   Out.oRunning := FALSE;
   Out.oHoming := FALSE;
   Out.oHomeRef := TRUE;
   Out.oServoPosOK := FALSE;
   Out.oErrorCode := -244;
   Out.oStatus := 0;
   Out.oActPosition := 113;
   Out.oManualListPos := 0;
   IO.ioManEnale := FALSE;
   IO.ioAutoEnale := FALSE;
   Spare.S[0] := 16#00;
   Spare.S[1] := 16#00;
   Spare.S[2] := 16#00;
   Spare.S[3] := 16#00;
   Spare.S[4] := 16#00;
   Spare.S[5] := 16#00;
   Spare.S[6] := 16#00;
   Spare.S[7] := 16#00;
   Spare.S[8] := 16#00;
   Spare.S[9] := 16#00;
   Spare.S[10] := 16#00;
   Spare.S[11] := 16#00;
   Spare.S[12] := 16#00;
   Spare.S[13] := 16#00;
   Spare.S[14] := 16#00;
   Spare.S[15] := 16#00;
   Spare.S[16] := 16#00;
   Spare.S[17] := 16#00;
   Spare.S[18] := 16#00;
   Spare.S[19] := 16#00;
   Spare.S[20] := 16#00;
   Spare.S[21] := 16#00;
   Spare.S[22] := 16#00;
   Spare.S[23] := 16#00;
   Spare.S[24] := 16#00;
   Spare.S[25] := 16#00;
   Spare.S[26] := 16#00;
   Spare.S[27] := 16#00;
   Spare.S[28] := 16#00;
   Spare.S[29] := 16#00;
   Spare.S[30] := 16#00;
   Spare.S[31] := 16#00;
   Spare.S[32] := 16#00;
   Spare.S[33] := 16#00;
   Spare.S[34] := 16#00;
   Spare.S[35] := 16#00;
   Spare.S[36] := 16#00;
   Spare.S[37] := 16#00;
   Spare.S[38] := 16#00;
   Spare.S[39] := 16#00;
   Spare.S[40] := 16#00;
   Spare.S[41] := 16#00;
   Spare.S[42] := 16#00;
   Spare.S[43] := 16#00;
   Spare.S[44] := 16#00;
   Spare.S[45] := 16#00;
   Spare.S[46] := 16#00;
   Spare.S[47] := 16#00;
   Spare.S[48] := 16#00;
   Spare.S[49] := 16#00;
   Spare.S[50] := 16#00;
   Spare.S[51] := 16#00;
   Spare.S[52] := 16#00;
   Spare.S[53] := 16#00;
   Spare.S[54] := 16#00;
   Spare.S[55] := 16#00;
   Spare.S[56] := 16#00;
   Spare.S[57] := 16#00;
   Spare.S[58] := 16#00;
   Spare.S[59] := 16#00;
   Spare.S[60] := 16#00;
   Spare.S[61] := 16#00;
   Spare.S[62] := 16#00;
   Spare.S[63] := 16#00;
   Spare.S[64] := 16#00;
   Spare.S[65] := 16#00;
   Spare.S[66] := 16#00;
   Spare.S[67] := 16#00;
   Spare.S[68] := 16#00;
   Spare.S[69] := 16#00;
   Spare.S[70] := 16#00;
   Spare.S[71] := 16#00;
   Spare.S[72] := 16#00;
   Spare.S[73] := 16#00;
   Spare.S[74] := 16#00;
   Spare.S[75] := 16#00;
   Spare.S[76] := 16#00;
   Spare.S[77] := 16#00;
   Spare.S[78] := 16#00;
   Spare.S[79] := 16#00;
   Spare.S[80] := 16#00;
   Spare.S[81] := 16#00;
   Spare.S[82] := 16#00;
   Spare.S[83] := 16#00;
   Spare.S[84] := 16#00;
   Spare.S[85] := 16#00;
   Spare.S[86] := 16#00;
   Spare.S[87] := 16#00;
   Spare.S[88] := 16#00;
   Spare.S[89] := 16#00;
   Spare.S[90] := 16#00;
   Spare.S[91] := 16#00;
   Spare.S[92] := 16#00;
   Spare.S[93] := 16#00;
   Spare.S[94] := 16#00;
   Spare.S[95] := 16#00;
   Spare.S[96] := 16#00;
   Spare.S[97] := 16#00;
   Spare.S[98] := 16#00;
   Spare.S[99] := 16#00;
   Spare.S[100] := 16#00;
   Manual.Index := 1;
   Manual.Pos[1].Pos := 0;
   Manual.Pos[1].Vel := 10000;
   Manual.Pos[2].Pos := 450000;
   Manual.Pos[2].Vel := 10000;
   Manual.Pos[3].Pos := 900000;
   Manual.Pos[3].Vel := 10000;
   Manual.Pos[4].Pos := 135000;
   Manual.Pos[4].Vel := 10000;
   Manual.Pos[5].Pos := 180000;
   Manual.Pos[5].Vel := 10000;
   Manual.Pos[6].Pos := 225000;
   Manual.Pos[6].Vel := 10000;
   Manual.Pos[7].Pos := 270000;
   Manual.Pos[7].Vel := 10000;
   Manual.Pos[8].Pos := 315000;
   Manual.Pos[8].Vel := 10000;
   Manual.Pos[9].Pos := 0;
   Manual.Pos[9].Vel := 0;
   Manual.Pos[10].Pos := 0;
   Manual.Pos[10].Vel := 0;
   Manual.Pos[11].Pos := 0;
   Manual.Pos[11].Vel := 0;
   Manual.Pos[12].Pos := 0;
   Manual.Pos[12].Vel := 0;
   Manual.Pos[13].Pos := 0;
   Manual.Pos[13].Vel := 0;
   Manual.Pos[14].Pos := 0;
   Manual.Pos[14].Vel := 0;
   Manual.Pos[15].Pos := 0;
   Manual.Pos[15].Vel := 0;
   Manual.Pos[16].Pos := 0;
   Manual.Pos[16].Vel := 0;
   Manual.Pos[17].Pos := 0;
   Manual.Pos[17].Vel := 0;
   Manual.Pos[18].Pos := 0;
   Manual.Pos[18].Vel := 0;
   Manual.Pos[19].Pos := 0;
   Manual.Pos[19].Vel := 0;
   Manual.Pos[20].Pos := 0;
   Manual.Pos[20].Vel := 0;
   Auto.Index := 1;
   Auto.Pos[1].Pos := 0;
   Auto.Pos[1].Vel := 10000;
   Auto.Pos[2].Pos := 450000;
   Auto.Pos[2].Vel := 10000;
   Auto.Pos[3].Pos := 900000;
   Auto.Pos[3].Vel := 10000;
   Auto.Pos[4].Pos := 135000;
   Auto.Pos[4].Vel := 10000;
   Auto.Pos[5].Pos := 180000;
   Auto.Pos[5].Vel := 10000;
   Auto.Pos[6].Pos := 225000;
   Auto.Pos[6].Vel := 10000;
   Auto.Pos[7].Pos := 270000;
   Auto.Pos[7].Vel := 10000;
   Auto.Pos[8].Pos := 315000;
   Auto.Pos[8].Vel := 10000;
   Auto.Pos[9].Pos := 0;
   Auto.Pos[9].Vel := 0;
   Auto.Pos[10].Pos := 0;
   Auto.Pos[10].Vel := 0;
   Auto.Pos[11].Pos := 0;
   Auto.Pos[11].Vel := 0;
   Auto.Pos[12].Pos := 0;
   Auto.Pos[12].Vel := 0;
   Auto.Pos[13].Pos := 0;
   Auto.Pos[13].Vel := 0;
   Auto.Pos[14].Pos := 0;
   Auto.Pos[14].Vel := 0;
   Auto.Pos[15].Pos := 0;
   Auto.Pos[15].Vel := 0;
   Auto.Pos[16].Pos := 0;
   Auto.Pos[16].Vel := 0;
   Auto.Pos[17].Pos := 0;
   Auto.Pos[17].Vel := 0;
   Auto.Pos[18].Pos := 0;
   Auto.Pos[18].Vel := 0;
   Auto.Pos[19].Pos := 0;
   Auto.Pos[19].Vel := 0;
   Auto.Pos[20].Pos := 0;
   Auto.Pos[20].Vel := 0;
   Interlock.Active := FALSE;
   Interlock.Case1 := TRUE;
   Interlock.Case2 := TRUE;
   Interlock.Case3 := FALSE;
   Interlock.Case4 := FALSE;
   Interlock.Case5 := FALSE;
   Interlock.Case6 := FALSE;
   Interlock.Case7 := FALSE;
   Interlock.Case8 := FALSE;
   Interlock.Case9 := FALSE;
   Interlock.Case10 := FALSE;
   PositionOk[1] := FALSE;
   PositionOk[2] := FALSE;
   PositionOk[3] := FALSE;
   PositionOk[4] := FALSE;
   PositionOk[5] := FALSE;
   PositionOk[6] := FALSE;
   PositionOk[7] := FALSE;
   PositionOk[8] := FALSE;
   PositionOk[9] := FALSE;
   PositionOk[10] := FALSE;
   PositionOk[11] := FALSE;
   PositionOk[12] := FALSE;
   PositionOk[13] := FALSE;
   PositionOk[14] := FALSE;
   PositionOk[15] := FALSE;
   PositionOk[16] := FALSE;
   PositionOk[17] := FALSE;
   PositionOk[18] := FALSE;
   PositionOk[19] := FALSE;
   PositionOk[20] := FALSE;
   Home_Pos."Home Pos Pls" := FALSE;
   Home_Pos."Arrow indication" := 0;
   Home_Pos."Process prompt" := 0;
   Home_Pos."Button prompt" := 0;

END_DATA_BLOCK

DATA_BLOCK "ServoV90_A4"
{ S7_Optimized_Access := 'FALSE' }
VERSION : 0.1
NON_RETAIN
   STRUCT 
      In : Struct
         iInterlock : Bool;
         "iManJog+" : Bool;
         "iManJog-" : Bool;
         iAutoStart : Bool;
         iHome : Bool;
         iCancelTask : Bool;
         iPauseTask : Bool;
         iManStart : Bool;
         iManListStart : Bool;
         iLimitSwitchActive : Bool;
         iLimitSoftActive : Bool;
         iRunningTimeout : Time;
         iHomingTimeout : Time;
         iAutoPosition : DInt;
         iAutoVelocity : Int;
         iManListPosition : DInt;
         iManListVelocity : Int;
         iManListNumber : Int;
         iManPosition : DInt;
         iManVelocity : Int;
         iMode : Int;
      END_STRUCT;
      Out : Struct
         oReady : Bool;
         oWarning : Bool;
         oError : Bool;
         oInterlock : Bool;
         oServoEnable : Bool;
         oRunning : Bool;
         oHoming : Bool;
         oHomeRef : Bool;
         oServoPosOK : Bool;
         oErrorCode : Int;
         oStatus : Int;
         oActPosition : DInt;
         oManualListPos : DInt;
      END_STRUCT;
      IO : Struct
         ioManEnale : Bool;
         ioAutoEnale : Bool;
      END_STRUCT;
      Spare : Struct
         S : Array[0..100] of Byte;
      END_STRUCT;
      Manual : Struct
         Index : Int;
         Pos : Array[1..20] of Struct
            Pos : DInt;
            Vel : Int;
         END_STRUCT;
      END_STRUCT;
      Auto : Struct
         Index : Int;
         Pos : Array[1..20] of Struct
            Pos : DInt;
            Vel : Int;
         END_STRUCT;
      END_STRUCT;
      Interlock : Struct
         Active : Bool;
         Case1 : Bool;
         Case2 : Bool;
         Case3 : Bool;
         Case4 : Bool;
         Case5 : Bool;
         Case6 : Bool;
         Case7 : Bool;
         Case8 : Bool;
         Case9 : Bool;
         Case10 : Bool;
      END_STRUCT;
      PositionOk : Array[1..20] of Bool;
      Home_Pos : Struct
         "Home Pos Pls" : Bool;
         "Arrow indication" : Int;
         "Process prompt" : Int;
         "Button prompt" : Int;
      END_STRUCT;
   END_STRUCT;


BEGIN
   In.iInterlock := TRUE;
   In."iManJog+" := FALSE;
   In."iManJog-" := FALSE;
   In.iAutoStart := FALSE;
   In.iHome := FALSE;
   In.iCancelTask := FALSE;
   In.iPauseTask := FALSE;
   In.iManStart := FALSE;
   In.iManListStart := FALSE;
   In.iLimitSwitchActive := TRUE;
   In.iLimitSoftActive := TRUE;
   In.iRunningTimeout := T#0MS;
   In.iHomingTimeout := T#0MS;
   In.iAutoPosition := 0;
   In.iAutoVelocity := 0;
   In.iManListPosition := 0;
   In.iManListVelocity := 0;
   In.iManListNumber := 0;
   In.iManPosition := 0;
   In.iManVelocity := 0;
   In.iMode := 0;
   Out.oReady := FALSE;
   Out.oWarning := FALSE;
   Out.oError := TRUE;
   Out.oInterlock := TRUE;
   Out.oServoEnable := FALSE;
   Out.oRunning := FALSE;
   Out.oHoming := FALSE;
   Out.oHomeRef := TRUE;
   Out.oServoPosOK := FALSE;
   Out.oErrorCode := -244;
   Out.oStatus := 0;
   Out.oActPosition := 260748;
   Out.oManualListPos := 3585;
   IO.ioManEnale := FALSE;
   IO.ioAutoEnale := FALSE;
   Spare.S[0] := 16#00;
   Spare.S[1] := 16#00;
   Spare.S[2] := 16#00;
   Spare.S[3] := 16#00;
   Spare.S[4] := 16#00;
   Spare.S[5] := 16#00;
   Spare.S[6] := 16#00;
   Spare.S[7] := 16#00;
   Spare.S[8] := 16#00;
   Spare.S[9] := 16#00;
   Spare.S[10] := 16#00;
   Spare.S[11] := 16#00;
   Spare.S[12] := 16#00;
   Spare.S[13] := 16#00;
   Spare.S[14] := 16#00;
   Spare.S[15] := 16#00;
   Spare.S[16] := 16#00;
   Spare.S[17] := 16#00;
   Spare.S[18] := 16#00;
   Spare.S[19] := 16#00;
   Spare.S[20] := 16#00;
   Spare.S[21] := 16#00;
   Spare.S[22] := 16#00;
   Spare.S[23] := 16#00;
   Spare.S[24] := 16#00;
   Spare.S[25] := 16#00;
   Spare.S[26] := 16#00;
   Spare.S[27] := 16#00;
   Spare.S[28] := 16#00;
   Spare.S[29] := 16#00;
   Spare.S[30] := 16#00;
   Spare.S[31] := 16#00;
   Spare.S[32] := 16#00;
   Spare.S[33] := 16#00;
   Spare.S[34] := 16#00;
   Spare.S[35] := 16#00;
   Spare.S[36] := 16#00;
   Spare.S[37] := 16#00;
   Spare.S[38] := 16#00;
   Spare.S[39] := 16#00;
   Spare.S[40] := 16#00;
   Spare.S[41] := 16#00;
   Spare.S[42] := 16#00;
   Spare.S[43] := 16#00;
   Spare.S[44] := 16#00;
   Spare.S[45] := 16#00;
   Spare.S[46] := 16#00;
   Spare.S[47] := 16#00;
   Spare.S[48] := 16#00;
   Spare.S[49] := 16#00;
   Spare.S[50] := 16#00;
   Spare.S[51] := 16#00;
   Spare.S[52] := 16#00;
   Spare.S[53] := 16#00;
   Spare.S[54] := 16#00;
   Spare.S[55] := 16#00;
   Spare.S[56] := 16#00;
   Spare.S[57] := 16#00;
   Spare.S[58] := 16#00;
   Spare.S[59] := 16#00;
   Spare.S[60] := 16#00;
   Spare.S[61] := 16#00;
   Spare.S[62] := 16#00;
   Spare.S[63] := 16#00;
   Spare.S[64] := 16#00;
   Spare.S[65] := 16#00;
   Spare.S[66] := 16#00;
   Spare.S[67] := 16#00;
   Spare.S[68] := 16#00;
   Spare.S[69] := 16#00;
   Spare.S[70] := 16#00;
   Spare.S[71] := 16#00;
   Spare.S[72] := 16#00;
   Spare.S[73] := 16#00;
   Spare.S[74] := 16#00;
   Spare.S[75] := 16#00;
   Spare.S[76] := 16#00;
   Spare.S[77] := 16#00;
   Spare.S[78] := 16#00;
   Spare.S[79] := 16#00;
   Spare.S[80] := 16#00;
   Spare.S[81] := 16#00;
   Spare.S[82] := 16#00;
   Spare.S[83] := 16#00;
   Spare.S[84] := 16#00;
   Spare.S[85] := 16#00;
   Spare.S[86] := 16#00;
   Spare.S[87] := 16#00;
   Spare.S[88] := 16#00;
   Spare.S[89] := 16#00;
   Spare.S[90] := 16#00;
   Spare.S[91] := 16#00;
   Spare.S[92] := 16#00;
   Spare.S[93] := 16#00;
   Spare.S[94] := 16#00;
   Spare.S[95] := 16#00;
   Spare.S[96] := 16#00;
   Spare.S[97] := 16#00;
   Spare.S[98] := 16#00;
   Spare.S[99] := 16#00;
   Spare.S[100] := 16#00;
   Manual.Index := 1;
   Manual.Pos[1].Pos := 3585;
   Manual.Pos[1].Vel := 10000;
   Manual.Pos[2].Pos := 48610;
   Manual.Pos[2].Vel := 10000;
   Manual.Pos[3].Pos := 93637;
   Manual.Pos[3].Vel := 10000;
   Manual.Pos[4].Pos := 138606;
   Manual.Pos[4].Vel := 10000;
   Manual.Pos[5].Pos := 183388;
   Manual.Pos[5].Vel := 10000;
   Manual.Pos[6].Pos := 228458;
   Manual.Pos[6].Vel := 10000;
   Manual.Pos[7].Pos := 273513;
   Manual.Pos[7].Vel := 10000;
   Manual.Pos[8].Pos := 318501;
   Manual.Pos[8].Vel := 10000;
   Manual.Pos[9].Pos := 0;
   Manual.Pos[9].Vel := 0;
   Manual.Pos[10].Pos := 0;
   Manual.Pos[10].Vel := 0;
   Manual.Pos[11].Pos := 0;
   Manual.Pos[11].Vel := 0;
   Manual.Pos[12].Pos := 0;
   Manual.Pos[12].Vel := 0;
   Manual.Pos[13].Pos := 0;
   Manual.Pos[13].Vel := 0;
   Manual.Pos[14].Pos := 0;
   Manual.Pos[14].Vel := 0;
   Manual.Pos[15].Pos := 0;
   Manual.Pos[15].Vel := 0;
   Manual.Pos[16].Pos := 0;
   Manual.Pos[16].Vel := 0;
   Manual.Pos[17].Pos := 0;
   Manual.Pos[17].Vel := 0;
   Manual.Pos[18].Pos := 0;
   Manual.Pos[18].Vel := 0;
   Manual.Pos[19].Pos := 0;
   Manual.Pos[19].Vel := 0;
   Manual.Pos[20].Pos := 0;
   Manual.Pos[20].Vel := 0;
   Auto.Index := 7;
   Auto.Pos[1].Pos := 3585;
   Auto.Pos[1].Vel := 10000;
   Auto.Pos[2].Pos := 48610;
   Auto.Pos[2].Vel := 10000;
   Auto.Pos[3].Pos := 93637;
   Auto.Pos[3].Vel := 10000;
   Auto.Pos[4].Pos := 138606;
   Auto.Pos[4].Vel := 10000;
   Auto.Pos[5].Pos := 183388;
   Auto.Pos[5].Vel := 10000;
   Auto.Pos[6].Pos := 228458;
   Auto.Pos[6].Vel := 10000;
   Auto.Pos[7].Pos := 273513;
   Auto.Pos[7].Vel := 10000;
   Auto.Pos[8].Pos := 318501;
   Auto.Pos[8].Vel := 10000;
   Auto.Pos[9].Pos := 0;
   Auto.Pos[9].Vel := 0;
   Auto.Pos[10].Pos := 0;
   Auto.Pos[10].Vel := 0;
   Auto.Pos[11].Pos := 0;
   Auto.Pos[11].Vel := 0;
   Auto.Pos[12].Pos := 0;
   Auto.Pos[12].Vel := 0;
   Auto.Pos[13].Pos := 0;
   Auto.Pos[13].Vel := 0;
   Auto.Pos[14].Pos := 0;
   Auto.Pos[14].Vel := 0;
   Auto.Pos[15].Pos := 0;
   Auto.Pos[15].Vel := 0;
   Auto.Pos[16].Pos := 0;
   Auto.Pos[16].Vel := 0;
   Auto.Pos[17].Pos := 0;
   Auto.Pos[17].Vel := 0;
   Auto.Pos[18].Pos := 0;
   Auto.Pos[18].Vel := 0;
   Auto.Pos[19].Pos := 0;
   Auto.Pos[19].Vel := 0;
   Auto.Pos[20].Pos := 0;
   Auto.Pos[20].Vel := 0;
   Interlock.Active := FALSE;
   Interlock.Case1 := TRUE;
   Interlock.Case2 := TRUE;
   Interlock.Case3 := FALSE;
   Interlock.Case4 := FALSE;
   Interlock.Case5 := FALSE;
   Interlock.Case6 := FALSE;
   Interlock.Case7 := FALSE;
   Interlock.Case8 := FALSE;
   Interlock.Case9 := FALSE;
   Interlock.Case10 := FALSE;
   PositionOk[1] := FALSE;
   PositionOk[2] := FALSE;
   PositionOk[3] := FALSE;
   PositionOk[4] := FALSE;
   PositionOk[5] := FALSE;
   PositionOk[6] := FALSE;
   PositionOk[7] := FALSE;
   PositionOk[8] := FALSE;
   PositionOk[9] := FALSE;
   PositionOk[10] := FALSE;
   PositionOk[11] := FALSE;
   PositionOk[12] := FALSE;
   PositionOk[13] := FALSE;
   PositionOk[14] := FALSE;
   PositionOk[15] := FALSE;
   PositionOk[16] := FALSE;
   PositionOk[17] := FALSE;
   PositionOk[18] := FALSE;
   PositionOk[19] := FALSE;
   PositionOk[20] := FALSE;
   Home_Pos."Home Pos Pls" := FALSE;
   Home_Pos."Arrow indication" := 0;
   Home_Pos."Process prompt" := 0;
   Home_Pos."Button prompt" := 0;

END_DATA_BLOCK

DATA_BLOCK "ServoV90_DeviceCtl"
{ S7_Optimized_Access := 'FALSE' }
VERSION : 0.1
   STRUCT 
      V90Servo : Array[1..4] of Struct
         i : Int;
         nError : Int;
         nWarning : Int;
         nPositionListNo : Int;
         Pos { S7_SetPoint := 'False'} : "PosList";
         Point : Array[0..39] of Struct
            Start : Bool;
            Achieve : Bool;
         END_STRUCT;
      END_STRUCT;
   END_STRUCT;


BEGIN
   V90Servo[1].nPositionListNo := 1;
   V90Servo[1].Pos.List[3].Vel := 0;
   V90Servo[1].Pos.List[4].Pos := 0;
   V90Servo[1].Pos.List[4].Vel := 0;
   V90Servo[1].Pos.List[5].Pos := 0;
   V90Servo[1].Pos.List[5].Vel := 0;
   V90Servo[1].Pos.List[6].Pos := 0;
   V90Servo[1].Pos.List[6].Vel := 0;
   V90Servo[1].Pos.List[7].Pos := 0;
   V90Servo[1].Pos.List[7].Vel := 0;
   V90Servo[1].Pos.List[8].Pos := 0;
   V90Servo[1].Pos.List[8].Vel := 0;
   V90Servo[1].Pos.List[9].Pos := 0;
   V90Servo[1].Pos.List[9].Vel := 0;
   V90Servo[1].Pos.List[10].Pos := 0;
   V90Servo[1].Pos.List[10].Vel := 0;
   V90Servo[1].Pos.List[11].Pos := 0;
   V90Servo[1].Pos.List[11].Vel := 0;
   V90Servo[1].Pos.List[12].Pos := 0;
   V90Servo[1].Pos.List[12].Vel := 0;
   V90Servo[1].Pos.List[13].Pos := 0;
   V90Servo[1].Pos.List[13].Vel := 0;
   V90Servo[1].Pos.List[14].Pos := 0;
   V90Servo[1].Pos.List[14].Vel := 0;
   V90Servo[1].Pos.List[15].Pos := 0;
   V90Servo[1].Pos.List[15].Vel := 0;
   V90Servo[1].Pos.List[16].Pos := 0;
   V90Servo[1].Pos.List[16].Vel := 0;
   V90Servo[1].Pos.List[17].Pos := 0;
   V90Servo[1].Pos.List[17].Vel := 0;
   V90Servo[1].Pos.List[18].Pos := 0;
   V90Servo[1].Pos.List[18].Vel := 0;
   V90Servo[1].Pos.List[19].Pos := 0;
   V90Servo[1].Pos.List[19].Vel := 0;
   V90Servo[2].nPositionListNo := 1;
   V90Servo[3].nPositionListNo := 1;
   V90Servo[4].nPositionListNo := 1;

END_DATA_BLOCK

DATA_BLOCK "ST10_DBInterface_Stopper"
{ S7_Optimized_Access := 'FALSE' }
VERSION : 0.1
NON_RETAIN
   STRUCT 
      Stopper : Array[1..50] of "UDT_StopperInterface";
   END_STRUCT;


BEGIN

END_DATA_BLOCK

DATA_BLOCK "ST10_StopperCtrl_DB"
{ S7_Optimized_Access := 'FALSE' }
VERSION : 0.1
NON_RETAIN
"ST10_StopperCtrl"

BEGIN

END_DATA_BLOCK

DATA_BLOCK "Pilz_fb_DB"
{ S7_Optimized_Access := 'FALSE' }
VERSION : 0.1
NON_RETAIN
"Pilz_fb"

BEGIN

END_DATA_BLOCK

DATA_BLOCK "PalletNGData"
{ S7_Optimized_Access := 'FALSE' }
VERSION : 0.1
NON_RETAIN
   STRUCT 
      LoadingNGPallet : Struct
         NG_1_1 : Bool;
         NG_1_2 : Bool;
         NG_1_3 : Bool;
         NG_1_4 : Bool;
         NG_1_5 : Bool;
         NG_2_1 : Bool;
         NG_2_2 : Bool;
         NG_2_3 : Bool;
         NG_2_4 : Bool;
         NG_2_5 : Bool;
         NG_3_1 : Bool;
         NG_3_2 : Bool;
         NG_3_3 : Bool;
         NG_3_4 : Bool;
         NG_3_5 : Bool;
         OpenFlag : Bool;
         Status_1 : Int;
         Status_2 : Int;
         Status_3 : Int;
         Ready_1 : Bool;
         Ready_2 : Bool;
         Ready_3 : Bool;
         Ready_4 : Bool;
         Ready_5 : Bool;
         Ready_6 : Bool;
         Ready : Bool;
         Interlock_1 : Array[1..10] of Bool;
         Interlock_2 : Array[1..10] of Bool;
         Interlock_3 : Array[1..10] of Bool;
         LockStatus : Int;
      END_STRUCT;
      UnLoadingNGPallet : Struct
         NG_1_1 : Bool;
         NG_1_2 : Bool;
         NG_1_3 : Bool;
         NG_1_4 : Bool;
         NG_1_5 : Bool;
         NG_2_1 : Bool;
         NG_2_2 : Bool;
         NG_2_3 : Bool;
         NG_2_4 : Bool;
         NG_2_5 : Bool;
         NG_3_1 : Bool;
         NG_3_2 : Bool;
         NG_3_3 : Bool;
         NG_3_4 : Bool;
         NG_3_5 : Bool;
         OpenFlag : Bool;
         Status_1 : Int;
         Status_2 : Int;
         Status_3 : Int;
         Ready_1 : Bool;
         Ready_2 : Bool;
         Ready_3 : Bool;
         Ready_4 : Bool;
         Ready_5 : Bool;
         Ready_6 : Bool;
         Ready : Bool;
         Interlock_1 : Array[1..10] of Bool;
         Interlock_2 : Array[1..10] of Bool;
         Interlock_3 : Array[1..10] of Bool;
         LockStatus : Int;
      END_STRUCT;
      P : Array[0..10] of Bool;
   END_STRUCT;


BEGIN

END_DATA_BLOCK

DATA_BLOCK "MotorContro_DB_12"
{ S7_Optimized_Access := 'TRUE' }
VERSION : 0.1
NON_RETAIN
"MotorContro"

BEGIN

END_DATA_BLOCK

DATA_BLOCK "MotorContro_DB_13"
{ S7_Optimized_Access := 'TRUE' }
VERSION : 0.1
NON_RETAIN
"MotorContro"

BEGIN

END_DATA_BLOCK

DATA_BLOCK "MotorContro_DB_14"
{ S7_Optimized_Access := 'TRUE' }
VERSION : 0.1
NON_RETAIN
"MotorContro"

BEGIN

END_DATA_BLOCK

DATA_BLOCK "MotorContro_DB_15"
{ S7_Optimized_Access := 'TRUE' }
VERSION : 0.1
NON_RETAIN
"MotorContro"

BEGIN

END_DATA_BLOCK

DATA_BLOCK "MotorContro_DB_16"
{ S7_Optimized_Access := 'TRUE' }
VERSION : 0.1
NON_RETAIN
"MotorContro"

BEGIN

END_DATA_BLOCK

DATA_BLOCK "MotorContro_DB_17"
{ S7_Optimized_Access := 'TRUE' }
VERSION : 0.1
NON_RETAIN
"MotorContro"

BEGIN

END_DATA_BLOCK

DATA_BLOCK "MotorContro_DB_3"
{ S7_Optimized_Access := 'TRUE' }
VERSION : 0.1
NON_RETAIN
"MotorContro"

BEGIN

END_DATA_BLOCK

DATA_BLOCK "MotorData"
{ S7_Optimized_Access := 'FALSE' }
VERSION : 0.1
NON_RETAIN
   STRUCT 
      Ton {InstructionName := 'TON_TIME'; LibVersion := '1.0'; S7_SetPoint := 'False'} : Array[0..50] of TON_TIME;
      P { S7_SetPoint := 'True'} : Array[0..50] of Bool;
      "Time" : Array[0..50] of Time;
   END_STRUCT;


BEGIN
   "Time"[0] := T#60s;
   "Time"[1] := T#60s;
   "Time"[2] := T#60s;
   "Time"[3] := T#60s;
   "Time"[4] := T#60s;
   "Time"[5] := T#60s;
   "Time"[6] := T#60s;
   "Time"[7] := T#60s;
   "Time"[8] := T#60s;
   "Time"[9] := T#60s;
   "Time"[10] := T#60s;
   "Time"[11] := T#60s;
   "Time"[12] := T#60s;
   "Time"[13] := T#60s;
   "Time"[14] := T#60s;
   "Time"[15] := T#60s;
   "Time"[16] := T#60s;
   "Time"[17] := T#60s;
   "Time"[18] := T#60s;
   "Time"[19] := T#60s;
   "Time"[20] := T#60s;
   "Time"[21] := T#60s;
   "Time"[22] := T#60s;
   "Time"[23] := T#60s;
   "Time"[24] := T#60s;
   "Time"[25] := T#60s;
   "Time"[26] := T#60s;
   "Time"[27] := T#60s;
   "Time"[28] := T#60s;
   "Time"[29] := T#60s;
   "Time"[30] := T#60s;
   "Time"[31] := T#60s;
   "Time"[32] := T#60s;
   "Time"[33] := T#60s;
   "Time"[34] := T#60s;
   "Time"[35] := T#60s;
   "Time"[36] := T#60s;
   "Time"[37] := T#60s;
   "Time"[38] := T#60s;
   "Time"[39] := T#60s;
   "Time"[40] := T#60s;
   "Time"[41] := T#60s;
   "Time"[42] := T#60s;
   "Time"[43] := T#60s;
   "Time"[44] := T#60s;
   "Time"[45] := T#60s;
   "Time"[46] := T#60s;
   "Time"[47] := T#60s;
   "Time"[48] := T#60s;
   "Time"[49] := T#60s;
   "Time"[50] := T#60s;

END_DATA_BLOCK

DATA_BLOCK "ST10_FB_S7connect_IDB"
{ S7_Optimized_Access := 'TRUE' }
VERSION : 0.1
NON_RETAIN
"ST10_FB_S7connect"

BEGIN

END_DATA_BLOCK

DATA_BLOCK "DB_maXYmosNC1"
{ S7_Optimized_Access := 'FALSE' }
VERSION : 0.1
NON_RETAIN
"KistlerPresser _FB"

BEGIN

END_DATA_BLOCK

DATA_BLOCK "KistlerPresser1_DB"
{ S7_Optimized_Access := 'FALSE' }
VERSION : 0.1
NON_RETAIN
   STRUCT 
      ShaftID : Array[0..50] of Char;
      HousingID_1 : Array[0..50] of Char;
      HousingID_2 : Array[0..50] of Char;
      Shaft : String[48];
      spare : String[48];
   END_STRUCT;


BEGIN
   spare := '46';

END_DATA_BLOCK

DATA_BLOCK "KistlerPressData2"
{ S7_Optimized_Access := 'FALSE' }
VERSION : 0.1
NON_RETAIN
   STRUCT 
      Spare : Struct
         Spare : Array[0..85] of Byte;
      END_STRUCT;
      Data : Struct
         EO01 : Struct
            "pvXMin-Y" : Real;
            "pvXMax-Y" : Real;
            "pvXMin-X" : Real;
            "pvXMax-X" : Real;
         END_STRUCT;
         EO02 : Struct
            "pvXMin-Y" : Real;
            "pvXMax-Y" : Real;
            "pvXMin-X" : Real;
            "pvXMax-X" : Real;
         END_STRUCT;
         EO03 : Struct
            "pvXMax-Y" : Real;
            "pvXMax-X" : Real;
         END_STRUCT;
      END_STRUCT;
      iWritePressData : Struct
         temp1 : Real;
      END_STRUCT;
      PressData1 : Struct
         pvBlock_X : Real;
         pvBlock_Y : Real;
      END_STRUCT;
      ManualPro : Int;
   END_STRUCT;


BEGIN

END_DATA_BLOCK

DATA_BLOCK "KistlerPresser2_DB"
{ S7_Optimized_Access := 'FALSE' }
VERSION : 0.1
NON_RETAIN
   STRUCT 
      ShaftID : Array[0..50] of Char;
      HousingID_1 : Array[0..50] of Char;
      HousingID_2 : Array[0..50] of Char;
      Shaft : String[48];
      spare : String[48];
   END_STRUCT;


BEGIN
   spare := '46';

END_DATA_BLOCK

ORGANIZATION_BLOCK "01_OB1"   // OB1, LAD, ProgramCycle
TITLE = "Main Program Sweep (Cycle)"
{ S7_Optimized_Access := 'FALSE' }
AUTHOR : STD
FAMILY : System
VERSION : 2.0
// 系统程序段无需改动
// stored: AutoNumber false, SetENOAutomatically false
   VAR_TEMP
      OB1_EV_CLASS : Byte;   // Bits 0-3 = 1 (Coming event), Bits 4-7 = 1 (Event class 1)
      OB1_SCAN_1 : Byte;   // 1 (Cold restart scan 1 of OB 1), 3 (Scan 2-n of OB 1)
      OB1_PRIORITY : Byte;   // Priority of OB Execution
      OB1_OB_NUMBR : Byte;   // 1 (Organization block 1, OB1)
      OB1_RESERVED_1 : Byte;   // Reserved for system
      OB1_RESERVED_2 : Byte;   // Reserved for system
      OB1_PREV_CYCLE : Int;   // Cycle time of previous OB1 scan (milliseconds)
      OB1_MIN_CYCLE : Int;   // Minimum cycle time of OB1 (milliseconds)
      OB1_MAX_CYCLE : Int;   // Maximum cycle time of OB1 (milliseconds)
      OB1_DATE_TIME : Date_And_Time;   // Date and time OB1 started
      i : Int;
   END_VAR
   VAR_TEMP   // added for the SCL form of the ladder/FBD networks
      _w1 : Bool;
   END_VAR
BEGIN

REGION Network 1: Normal ON & OFF
   // 系统程序段
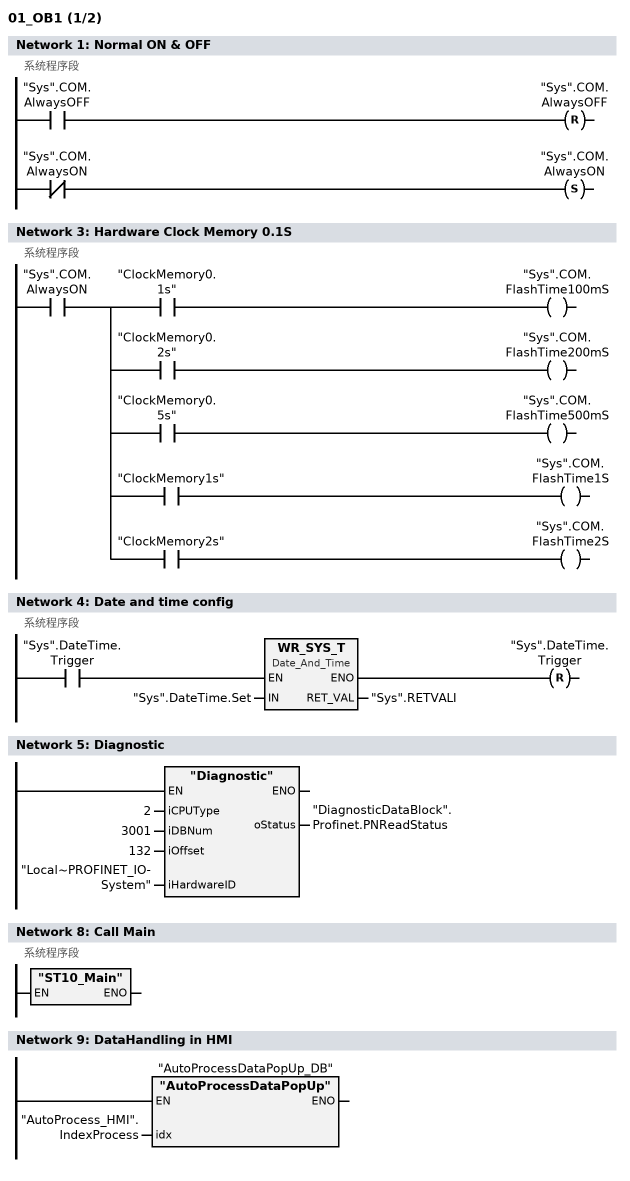
   RUNG wire#powerrail
      Contact( "Sys".COM.AlwaysOFF )
      R_Coil( "Sys".COM.AlwaysOFF )
   END_RUNG
   RUNG wire#powerrail
      I_Contact( "Sys".COM.AlwaysON )
      S_Coil( "Sys".COM.AlwaysON )
   END_RUNG
   // the same network as SCL:
   IF "Sys".COM.AlwaysOFF THEN "Sys".COM.AlwaysOFF := FALSE; END_IF;
   IF NOT "Sys".COM.AlwaysON THEN "Sys".COM.AlwaysON := TRUE; END_IF;
END_REGION

REGION Network 2 (SCL): ScanTime
   // System Function don't modify
   "Sys".ScanTime.CyclePrevious := #OB1_PREV_CYCLE;
   "Sys".ScanTime.CycleMin := #OB1_MIN_CYCLE;
   "Sys".ScanTime.CycleMax := #OB1_MAX_CYCLE;
END_REGION

REGION Network 3: Hardware Clock Memory 0.1S
   // 系统程序段
   RUNG wire#powerrail
      Contact( "Sys".COM.AlwaysON )
      wire#w1
      Contact( "ClockMemory0.1s" )
      Coil( "Sys".COM.FlashTime100mS )
   END_RUNG
   RUNG wire#w1
      Contact( "ClockMemory0.2s" )
      Coil( "Sys".COM.FlashTime200mS )
   END_RUNG
   RUNG wire#w1
      Contact( "ClockMemory0.5s" )
      Coil( "Sys".COM.FlashTime500mS )
   END_RUNG
   RUNG wire#w1
      Contact( "ClockMemory1s" )
      Coil( "Sys".COM.FlashTime1S )
   END_RUNG
   RUNG wire#w1
      Contact( "ClockMemory2s" )
      Coil( "Sys".COM.FlashTime2S )
   END_RUNG
   // the same network as SCL:
   "Sys".COM.FlashTime100mS := "Sys".COM.AlwaysON AND "ClockMemory0.1s";
   "Sys".COM.FlashTime200mS := "Sys".COM.AlwaysON AND "ClockMemory0.2s";
   "Sys".COM.FlashTime500mS := "Sys".COM.AlwaysON AND "ClockMemory0.5s";
   "Sys".COM.FlashTime1S := "Sys".COM.AlwaysON AND "ClockMemory1s";
   "Sys".COM.FlashTime2S := "Sys".COM.AlwaysON AND "ClockMemory2s";
END_REGION

REGION Network 4: Date and time config
   // 系统程序段
   RUNG wire#powerrail
      Contact( "Sys".DateTime.Trigger )
      { S7_Templates := "date_type := Date_And_Time" } WR_SYS_T(IN := "Sys".DateTime.Set, RET_VAL => "Sys".RETVALI)
      R_Coil( "Sys".DateTime.Trigger )
   END_RUNG
   // the same network as SCL:
   "Sys".RETVALI := WR_SYS_T(EN := "Sys".DateTime.Trigger, IN := "Sys".DateTime.Set, ENO => #_w1);
   IF #_w1 THEN "Sys".DateTime.Trigger := FALSE; END_IF;
END_REGION

REGION Network 5: Diagnostic
   RUNG wire#powerrail
      "Diagnostic"(iCPUType := 2, iDBNum := 3001, iOffset := 132, iHardwareID := "Local~PROFINET_IO-System", oStatus => "DiagnosticDataBlock".Profinet.PNReadStatus)
   END_RUNG
   // the same network as SCL:
   "Diagnostic"(iCPUType := 2,
                iDBNum := 3001,
                iOffset := 132,
                iHardwareID := "Local~PROFINET_IO-System",
                oStatus => "DiagnosticDataBlock".Profinet.PNReadStatus);
END_REGION

REGION Network 6 (SCL): Win
       "ST10_GeneralData".HMI.Win.WinBullfer := 0;
       FOR #i := 1 TO 10 DO
           "ST10_GeneralData".HMI.Win.WinBullfer := "ST10_GeneralData".HMI.Win.WinBullfer + "ST10_GeneralData".HMI.Win."10x弹窗"[#i] * 11 +"ST10_GeneralData".HMI.Win."20x弹窗"[2] * 21 +"ST10_GeneralData".HMI.Win."30x弹窗"[#i] * 31 +"ST10_GeneralData".HMI.Win."40x弹窗"[#i] * 41;
       END_FOR;
       "ST10_GeneralData".HMI.Win.WinBullfer := ABS("ST10_GeneralData".HMI.Win.WinBullfer);
       "ST10_GeneralData".HMI.Win.TON[1](IN := "ST10_GeneralData".HMI.Win.Win <> "ST10_GeneralData".HMI.Win.WinBullfer,
                          PT := T#0.5S);
   IF "ST10_GeneralData".HMI.Win.TON[1].Q THEN
       "ST10_GeneralData".HMI.Win.Win := "ST10_GeneralData".HMI.Win.WinBullfer;
       END_IF;
END_REGION

REGION Network 7: MES_Shopworx
END_REGION

REGION Network 8: Call Main
   // 系统程序段
   RUNG wire#powerrail
      "ST10_Main"()
   END_RUNG
   // the same network as SCL:
   "ST10_Main"();
END_REGION

REGION Network 9: DataHandling in HMI
   RUNG wire#powerrail
      "AutoProcessDataPopUp_DB"(idx := "AutoProcess_HMI".IndexProcess)
   END_RUNG
   // the same network as SCL:
   "AutoProcessDataPopUp_DB"(idx := "AutoProcess_HMI".IndexProcess);   // "AutoProcessDataPopUp"
END_REGION

REGION Network 10: 上电初始化设备模式_手动模式 / Power-on Initialization Device Mode _ Manual mode
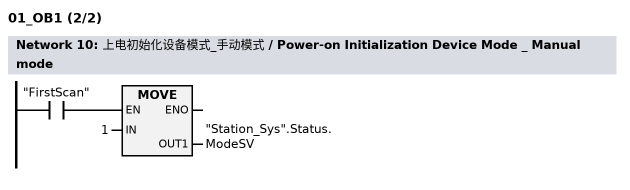
   RUNG wire#powerrail
      Contact( "FirstScan" )
      Move(in := 1, out1 => "Station_Sys".Status.ModeSV)
   END_RUNG
   // the same network as SCL:
   IF "FirstScan" THEN "Station_Sys".Status.ModeSV := 1; END_IF;
END_REGION
END_ORGANIZATION_BLOCK

FUNCTION "Diagnostic" : Void
{ S7_Optimized_Access := 'FALSE' }
AUTHOR : STD
FAMILY : RCS
VERSION : 18.0
   VAR_INPUT 
      iCPUType : Int;
      iDBNum : Word;
      iOffset : Int;
      iHardwareID : HW_IOSYSTEM;
   END_VAR

   VAR_OUTPUT 
      oStatus : Int;
   END_VAR

   VAR_TEMP 
      RDSRet : Struct
         Busy : Bool;
         Header : Struct
            Length : Word;
            Number : Word;
         END_STRUCT;
      END_STRUCT;
      retInt : Int;
      SSL : Struct
         SSID : Word;
         Index : Word;
         Length : Int;
      END_STRUCT;
      DR : Any;
      DRS AT DR : Struct
         SyntaxID : Byte;
         DataType : Byte;
         RepetitionFactor : Int;
         DB_Number : Word;
         MemoryAreaAddress : DWord;
      END_STRUCT;
   END_VAR


BEGIN
	
	(*############################################################
	   RUHLAMAT SUZHOU ELEC.STD.
	   Copyright (c) 2017. All rights reserved.    
	
	   NAME OF FUNCTION BLOCK:         Diagnostic
	   VERSION NUMBER:                 V3.0
	   COMPOSER:                       Ming.Jiang
	   
	   CreateDate:                    16.Nov.2016
	   ----------------------------------------------------------
	   Interface description:
	   IN:
	       "iCPUType"
	       iDBNum
	       iOffset
	       iHardwareID
	
	   INOUT:
	   OUT:
	       oStatus
	
	   ----------------------------------------------------------
	   #RET_VALUE:
	  
	   #Alert Value:
	  
	   ----------------------------------------------------------
	   Date           Name      Version           Activity                                                                              
	   28.Nov.2016    JM        V3.0              add alarm
	   
	############################################################*)
	IF #iCPUType = 0 OR #iDBNum = 0 THEN
	    ENO := 0;
	    RETURN;
	ELSE
	    IF #iCPUType=2 THEN
	        GOTO PN;
	    ELSIF #iCPUType=1 THEN
	        ;
	    ELSE
	        ENO := 0;
	        RETURN;
	    END_IF;
	    #DRS.SyntaxID := 16#10;
	    #DRS.DataType := 16#02;
	    #DRS.RepetitionFactor := 128;
	    #DRS.DB_Number := #iDBNum;
	    #DRS.MemoryAreaAddress := 16#8400_0000 OR (SHL(IN := INT_TO_DWORD(#iOffset), N := 3));
	    #oStatus := DeviceStates(LADDR := #iHardwareID, MODE := 2, STATE := #DR);
	PN:
	    #DRS.SyntaxID := 16#10;
	    #DRS.DataType := 16#02;
	    #DRS.RepetitionFactor := 128;
	    #DRS.DB_Number := #iDBNum;
	    #DRS.MemoryAreaAddress := 16#8400_0000 OR (SHL(IN := INT_TO_DWORD(#iOffset), N := 3));
	    #oStatus := DeviceStates(LADDR := #iHardwareID, MODE := 2, STATE := #DR);
	    // orginise interface data 
	    ENO := 1;
	    RETURN;
	END_IF;
	
	
	
	
END_FUNCTION

FUNCTION "ST10_Main" : Void   // FC1050, LAD
{ S7_Optimized_Access := 'FALSE' }
// stored: AutoNumber false, SetENOAutomatically false
BEGIN

REGION Network 1
   // 系统功能组调用部分
   // 1.该部分用户可以自己根据系统的组成将需要的功能块调用写在该部分
   // 2.该部分禁止与系统功能无关的程序在此处调用
END_REGION

NETWORK
TITLE = XXXX=====Station Relation/工位相关 =====StartXXXXX / XXXX=====Station Relation/Station correlation =====StartXXXXX

REGION Network 3: input /输入
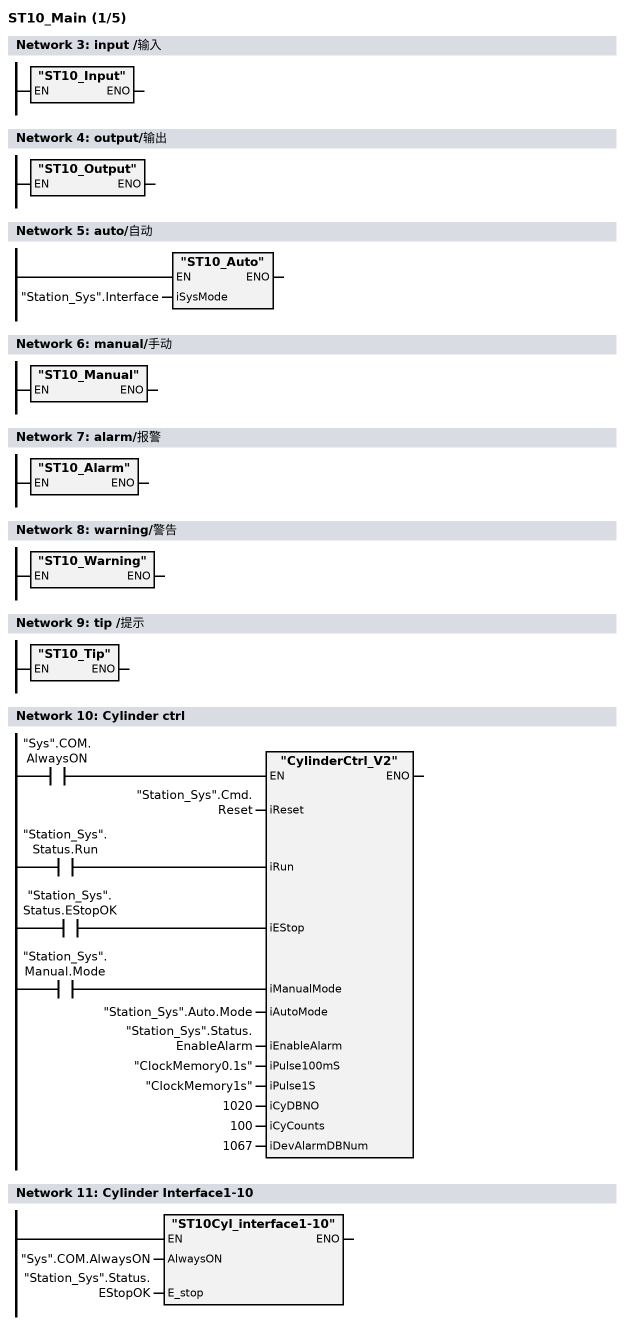
   RUNG wire#powerrail
      "ST10_Input"()
   END_RUNG
   // the same network as SCL:
   "ST10_Input"();
END_REGION

REGION Network 4: output/输出
   RUNG wire#powerrail
      "ST10_Output"()
   END_RUNG
   // the same network as SCL:
   "ST10_Output"();
END_REGION

REGION Network 5: auto/自动
   RUNG wire#powerrail
      "ST10_Auto"(iSysMode := "Station_Sys".Interface)
   END_RUNG
   // the same network as SCL:
   "ST10_Auto"(iSysMode := "Station_Sys".Interface);
END_REGION

REGION Network 6: manual/手动
   RUNG wire#powerrail
      "ST10_Manual"()
   END_RUNG
   // the same network as SCL:
   "ST10_Manual"();
END_REGION

REGION Network 7: alarm/报警
   RUNG wire#powerrail
      "ST10_Alarm"()
   END_RUNG
   // the same network as SCL:
   "ST10_Alarm"();
END_REGION

REGION Network 8: warning/警告
   RUNG wire#powerrail
      "ST10_Warning"()
   END_RUNG
   // the same network as SCL:
   "ST10_Warning"();
END_REGION

REGION Network 9: tip /提示
   RUNG wire#powerrail
      "ST10_Tip"()
   END_RUNG
   // the same network as SCL:
   "ST10_Tip"();
END_REGION

REGION Network 10: Cylinder ctrl
   RUNG wire#powerrail
      Contact( "Sys".COM.AlwaysON )
      "CylinderCtrl_V2"(iRun := wire#w1, iEStop := wire#w2, iManualMode := wire#w3, iReset := "Station_Sys".Cmd.Reset, iAutoMode := "Station_Sys".Auto.Mode, iEnableAlarm := "Station_Sys".Status.EnableAlarm, iPulse100mS := "ClockMemory0.1s", iPulse1S := "ClockMemory1s", iCyDBNO := 1020, iCyCounts := 100, iDevAlarmDBNum := 1067)
   END_RUNG
   RUNG wire#powerrail
      Contact( "Station_Sys".Status.Run )
   END_RUNG wire#w1
   RUNG wire#powerrail
      Contact( "Station_Sys".Status.EStopOK )
   END_RUNG wire#w2
   RUNG wire#powerrail
      Contact( "Station_Sys".Manual.Mode )
   END_RUNG wire#w3
   // the same network as SCL:
   IF "Sys".COM.AlwaysON THEN
       "CylinderCtrl_V2"(iReset := "Station_Sys".Cmd.Reset,
                         iRun := "Station_Sys".Status.Run,
                         iEStop := "Station_Sys".Status.EStopOK,
                         iManualMode := "Station_Sys".Manual.Mode,
                         iAutoMode := "Station_Sys".Auto.Mode,
                         iEnableAlarm := "Station_Sys".Status.EnableAlarm,
                         iPulse100mS := "ClockMemory0.1s",
                         iPulse1S := "ClockMemory1s",
                         iCyDBNO := 1020,
                         iCyCounts := 100,
                         iDevAlarmDBNum := 1067);
   END_IF;
END_REGION

REGION Network 11: Cylinder Interface1-10
   RUNG wire#powerrail
      "ST10Cyl_interface1-10"(AlwaysON := "Sys".COM.AlwaysON, E_stop := "Station_Sys".Status.EStopOK)
   END_RUNG
   // the same network as SCL:
   "ST10Cyl_interface1-10"(AlwaysON := "Sys".COM.AlwaysON, E_stop := "Station_Sys".Status.EStopOK);
END_REGION

REGION Network 12: Cylinder Interface11-20
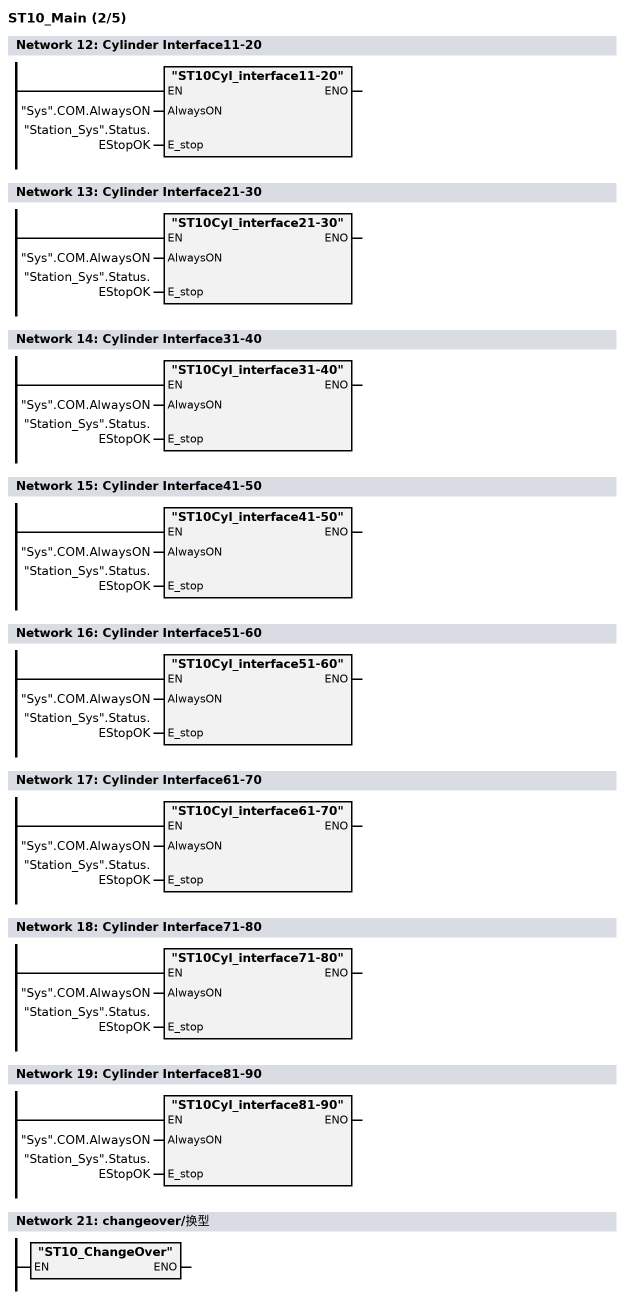
   RUNG wire#powerrail
      "ST10Cyl_interface11-20"(AlwaysON := "Sys".COM.AlwaysON, E_stop := "Station_Sys".Status.EStopOK)
   END_RUNG
   // the same network as SCL:
   "ST10Cyl_interface11-20"(AlwaysON := "Sys".COM.AlwaysON, E_stop := "Station_Sys".Status.EStopOK);
END_REGION

REGION Network 13: Cylinder Interface21-30
   RUNG wire#powerrail
      "ST10Cyl_interface21-30"(AlwaysON := "Sys".COM.AlwaysON, E_stop := "Station_Sys".Status.EStopOK)
   END_RUNG
   // the same network as SCL:
   "ST10Cyl_interface21-30"(AlwaysON := "Sys".COM.AlwaysON, E_stop := "Station_Sys".Status.EStopOK);
END_REGION

REGION Network 14: Cylinder Interface31-40
   RUNG wire#powerrail
      "ST10Cyl_interface31-40"(AlwaysON := "Sys".COM.AlwaysON, E_stop := "Station_Sys".Status.EStopOK)
   END_RUNG
   // the same network as SCL:
   "ST10Cyl_interface31-40"(AlwaysON := "Sys".COM.AlwaysON, E_stop := "Station_Sys".Status.EStopOK);
END_REGION

REGION Network 15: Cylinder Interface41-50
   RUNG wire#powerrail
      "ST10Cyl_interface41-50"(AlwaysON := "Sys".COM.AlwaysON, E_stop := "Station_Sys".Status.EStopOK)
   END_RUNG
   // the same network as SCL:
   "ST10Cyl_interface41-50"(AlwaysON := "Sys".COM.AlwaysON, E_stop := "Station_Sys".Status.EStopOK);
END_REGION

REGION Network 16: Cylinder Interface51-60
   RUNG wire#powerrail
      "ST10Cyl_interface51-60"(AlwaysON := "Sys".COM.AlwaysON, E_stop := "Station_Sys".Status.EStopOK)
   END_RUNG
   // the same network as SCL:
   "ST10Cyl_interface51-60"(AlwaysON := "Sys".COM.AlwaysON, E_stop := "Station_Sys".Status.EStopOK);
END_REGION

REGION Network 17: Cylinder Interface61-70
   RUNG wire#powerrail
      "ST10Cyl_interface61-70"(AlwaysON := "Sys".COM.AlwaysON, E_stop := "Station_Sys".Status.EStopOK)
   END_RUNG
   // the same network as SCL:
   "ST10Cyl_interface61-70"(AlwaysON := "Sys".COM.AlwaysON, E_stop := "Station_Sys".Status.EStopOK);
END_REGION

REGION Network 18: Cylinder Interface71-80
   RUNG wire#powerrail
      "ST10Cyl_interface71-80"(AlwaysON := "Sys".COM.AlwaysON, E_stop := "Station_Sys".Status.EStopOK)
   END_RUNG
   // the same network as SCL:
   "ST10Cyl_interface71-80"(AlwaysON := "Sys".COM.AlwaysON, E_stop := "Station_Sys".Status.EStopOK);
END_REGION

REGION Network 19: Cylinder Interface81-90
   RUNG wire#powerrail
      "ST10Cyl_interface81-90"(AlwaysON := "Sys".COM.AlwaysON, E_stop := "Station_Sys".Status.EStopOK)
   END_RUNG
   // the same network as SCL:
   "ST10Cyl_interface81-90"(AlwaysON := "Sys".COM.AlwaysON, E_stop := "Station_Sys".Status.EStopOK);
END_REGION

REGION Network 21: changeover/换型
   RUNG wire#powerrail
      "ST10_ChangeOver"()
   END_RUNG
   // the same network as SCL:
   "ST10_ChangeOver"();
END_REGION

REGION Network 22: Device
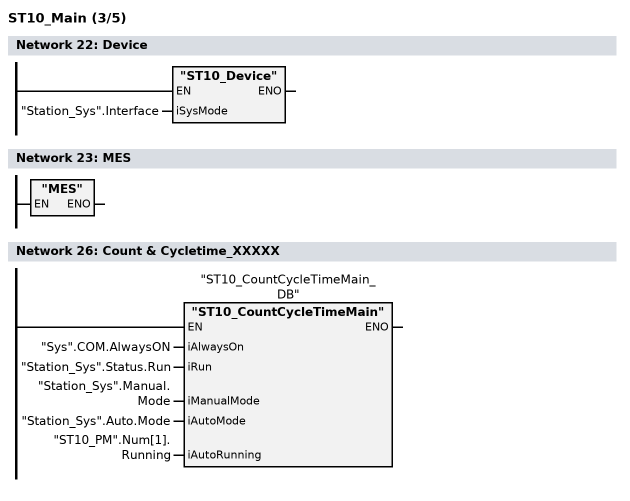
   RUNG wire#powerrail
      "ST10_Device"(iSysMode := "Station_Sys".Interface)
   END_RUNG
   // the same network as SCL:
   "ST10_Device"(iSysMode := "Station_Sys".Interface);
END_REGION

REGION Network 23: MES
   RUNG wire#powerrail
      "MES"()
   END_RUNG
   // the same network as SCL:
   "MES"();
END_REGION

REGION Network 24: =====System Function related information Section =====Start
END_REGION

NETWORK
TITLE = SystemFunction IO

REGION Network 26: Count & Cycletime_XXXXX
   RUNG wire#powerrail
      "ST10_CountCycleTimeMain_DB"(iAlwaysOn := "Sys".COM.AlwaysON, iRun := "Station_Sys".Status.Run, iManualMode := "Station_Sys".Manual.Mode, iAutoMode := "Station_Sys".Auto.Mode, iAutoRunning := "ST10_PM".Num[1].Running)
   END_RUNG
   // the same network as SCL:
   "ST10_CountCycleTimeMain_DB"(iAlwaysOn := "Sys".COM.AlwaysON,   // "ST10_CountCycleTimeMain"
                           iRun := "Station_Sys".Status.Run,
                           iManualMode := "Station_Sys".Manual.Mode,
                           iAutoMode := "Station_Sys".Auto.Mode,
                           iAutoRunning := "ST10_PM".Num[1].Running);
END_REGION

REGION Network 27: System mode
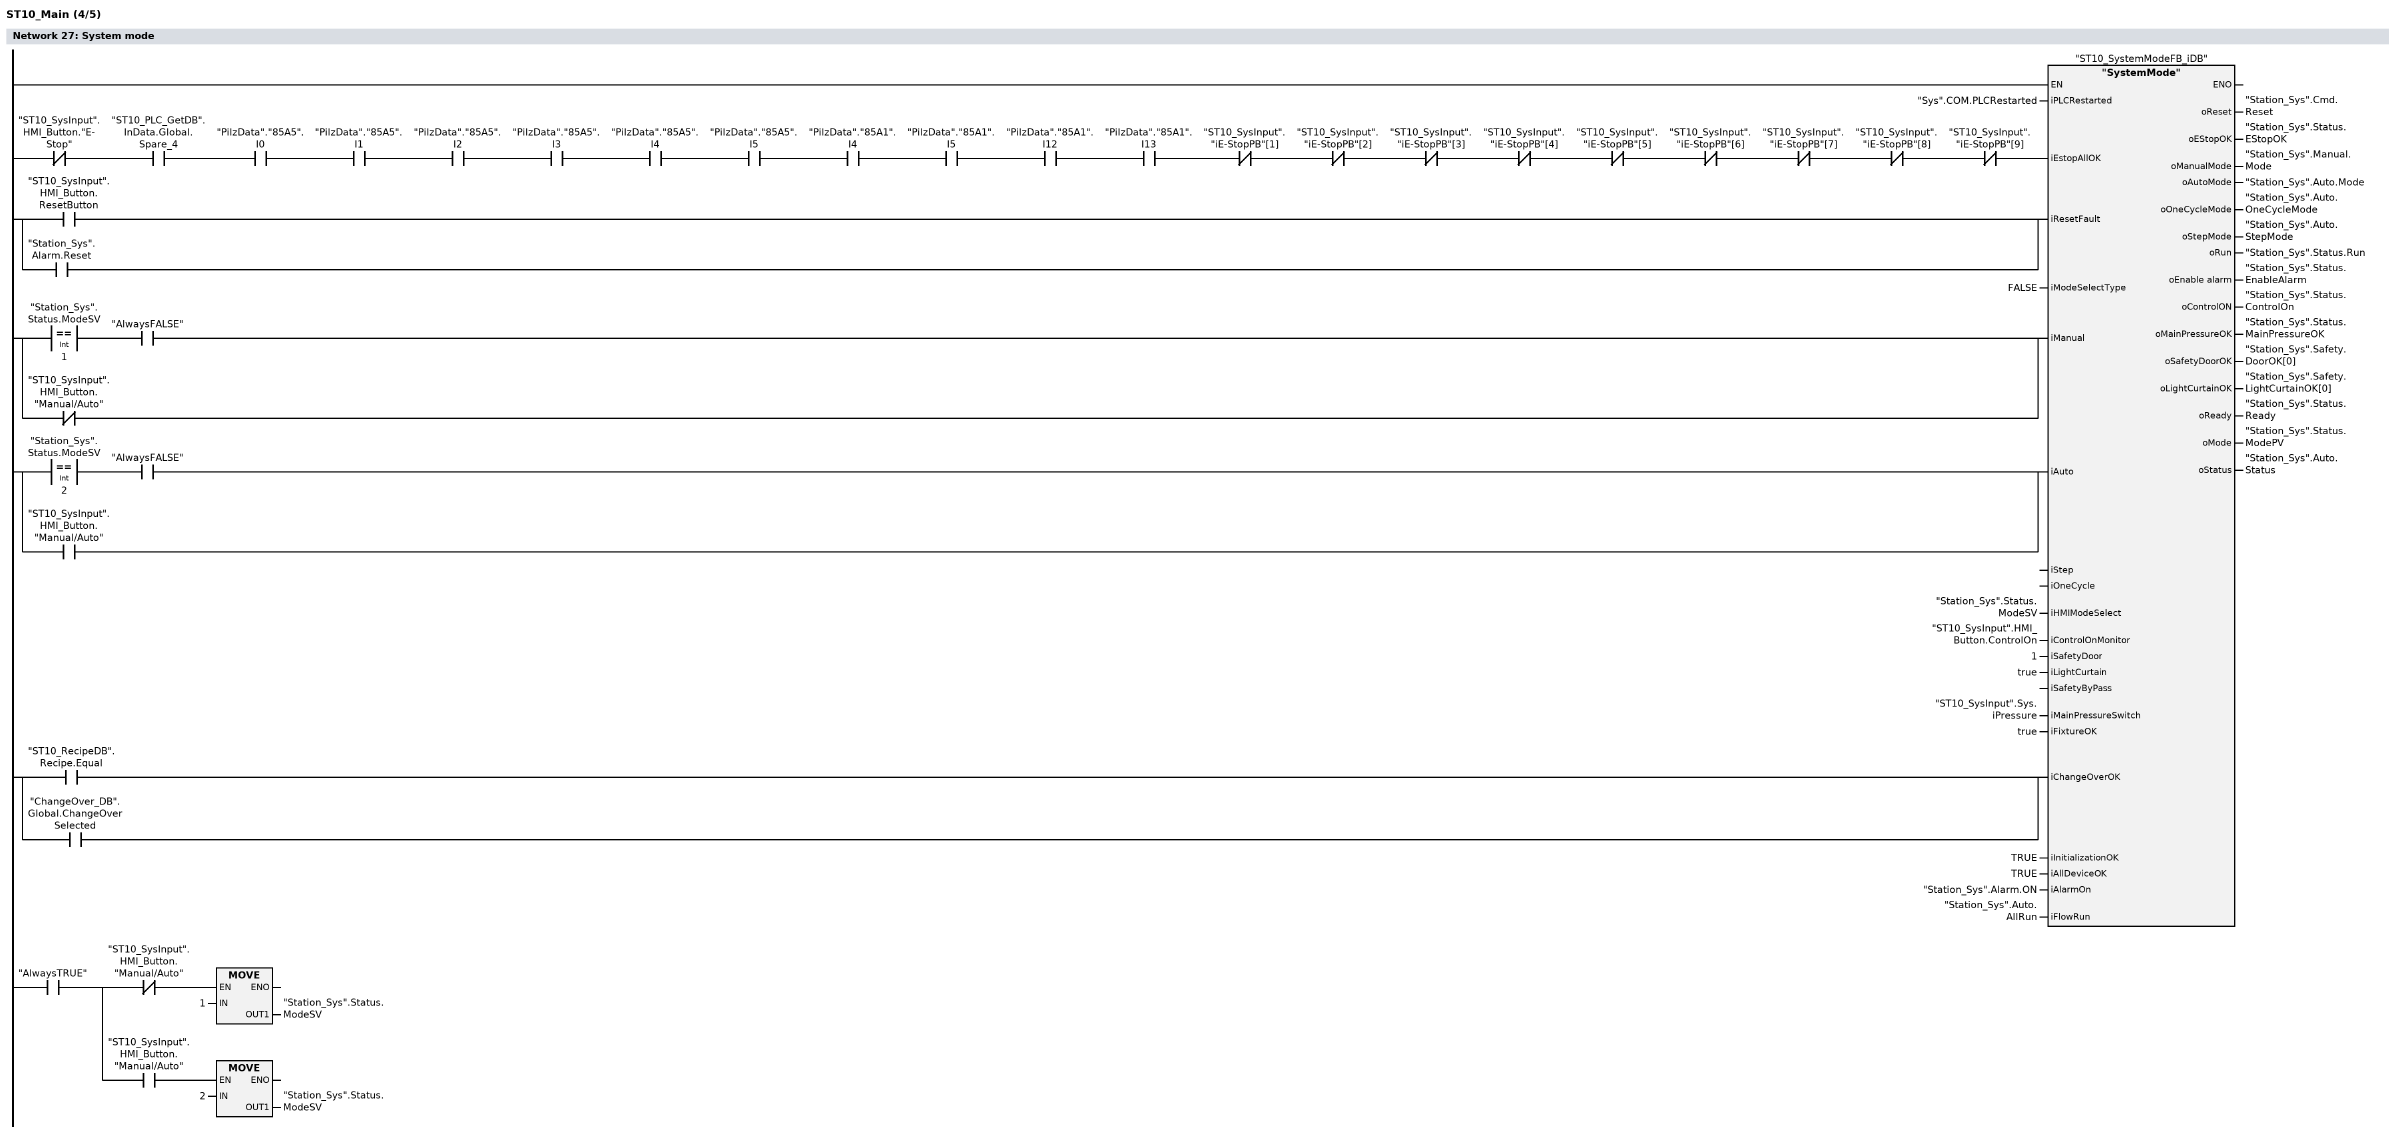
   RUNG wire#powerrail
      "ST10_SystemModeFB_iDB"(iEstopAllOK := wire#w1, iResetFault := wire#w2, iManual := wire#w3, iAuto := wire#w4, iChangeOverOK := wire#w5, iPLCRestarted := "Sys".COM.PLCRestarted, iModeSelectType := FALSE, iStep :=, iOneCycle :=, iHMIModeSelect := "Station_Sys".Status.ModeSV, iControlOnMonitor := "ST10_SysInput".HMI_Button.ControlOn, iSafetyDoor := 1, iLightCurtain := true, iSafetyByPass :=, iMainPressureSwitch := "ST10_SysInput".Sys.iPressure, iFixtureOK := true, iInitializationOK := TRUE, iAllDeviceOK := TRUE, iAlarmOn := "Station_Sys".Alarm.ON, iFlowRun := "Station_Sys".Auto.AllRun, oReset => "Station_Sys".Cmd.Reset, oEStopOK => "Station_Sys".Status.EStopOK, oManualMode => "Station_Sys".Manual.Mode, oAutoMode => "Station_Sys".Auto.Mode, oOneCycleMode => "Station_Sys".Auto.OneCycleMode, oStepMode => "Station_Sys".Auto.StepMode, oRun => "Station_Sys".Status.Run, "oEnable alarm" => "Station_Sys".Status.EnableAlarm, oControlON => "Station_Sys".Status.ControlOn, oMainPressureOK => "Station_Sys".Status.MainPressureOK, oSafetyDoorOK => "Station_Sys".Safety.DoorOK[0], oLightCurtainOK => "Station_Sys".Safety.LightCurtainOK[0], oReady => "Station_Sys".Status.Ready, oMode => "Station_Sys".Status.ModePV, oStatus => "Station_Sys".Auto.Status)
   END_RUNG
   RUNG wire#powerrail
      I_Contact( "ST10_SysInput".HMI_Button."E-Stop" )
      Contact( "ST10_PLC_GetDB".InData.Global.Spare_4 )
      Contact( "PilzData"."85A5".I0 )
      Contact( "PilzData"."85A5".I1 )
      Contact( "PilzData"."85A5".I2 )
      Contact( "PilzData"."85A5".I3 )
      Contact( "PilzData"."85A5".I4 )
      Contact( "PilzData"."85A5".I5 )
      Contact( "PilzData"."85A1".I4 )
      Contact( "PilzData"."85A1".I5 )
      Contact( "PilzData"."85A1".I12 )
      Contact( "PilzData"."85A1".I13 )
      I_Contact( "ST10_SysInput"."iE-StopPB"[1] )
      I_Contact( "ST10_SysInput"."iE-StopPB"[2] )
      I_Contact( "ST10_SysInput"."iE-StopPB"[3] )
      I_Contact( "ST10_SysInput"."iE-StopPB"[4] )
      I_Contact( "ST10_SysInput"."iE-StopPB"[5] )
      I_Contact( "ST10_SysInput"."iE-StopPB"[6] )
      I_Contact( "ST10_SysInput"."iE-StopPB"[7] )
      I_Contact( "ST10_SysInput"."iE-StopPB"[8] )
      I_Contact( "ST10_SysInput"."iE-StopPB"[9] )
   END_RUNG wire#w1
   RUNG wire#powerrail
      Contact( "ST10_SysInput".HMI_Button.ResetButton )
   END_RUNG wire#w2
   RUNG wire#powerrail
      Contact( "Station_Sys".Alarm.Reset )
   END_RUNG wire#w2
   RUNG wire#powerrail
      { S7_Templates := "SrcType := Int" } EQ_Contact(in1 := "Station_Sys".Status.ModeSV, in2 := 1)
      Contact( "AlwaysFALSE" )
   END_RUNG wire#w3
   RUNG wire#powerrail
      I_Contact( "ST10_SysInput".HMI_Button."Manual/Auto" )
   END_RUNG wire#w3
   RUNG wire#powerrail
      { S7_Templates := "SrcType := Int" } EQ_Contact(in1 := "Station_Sys".Status.ModeSV, in2 := 2)
      Contact( "AlwaysFALSE" )
   END_RUNG wire#w4
   RUNG wire#powerrail
      Contact( "ST10_SysInput".HMI_Button."Manual/Auto" )
   END_RUNG wire#w4
   RUNG wire#powerrail
      Contact( "ST10_RecipeDB".Recipe.Equal )
   END_RUNG wire#w5
   RUNG wire#powerrail
      Contact( "ChangeOver_DB".Global.ChangeOverSelected )
   END_RUNG wire#w5
   RUNG wire#powerrail
      Contact( "AlwaysTRUE" )
      wire#w6
      I_Contact( "ST10_SysInput".HMI_Button."Manual/Auto" )
      Move(in := 1, out1 => "Station_Sys".Status.ModeSV)
   END_RUNG
   RUNG wire#w6
      Contact( "ST10_SysInput".HMI_Button."Manual/Auto" )
      Move(in := 2, out1 => "Station_Sys".Status.ModeSV)
   END_RUNG
   // the same network as SCL:
   "ST10_SystemModeFB_iDB"(iPLCRestarted := "Sys".COM.PLCRestarted,   // "SystemMode"
                           iEstopAllOK := NOT "ST10_SysInput".HMI_Button."E-Stop" AND "ST10_PLC_GetDB".InData.Global.Spare_4 AND "PilzData"."85A5".I0 AND "PilzData"."85A5".I1 AND "PilzData"."85A5".I2 AND "PilzData"."85A5".I3 AND "PilzData"."85A5".I4 AND "PilzData"."85A5".I5 AND "PilzData"."85A1".I4 AND "PilzData"."85A1".I5 AND "PilzData"."85A1".I12 AND "PilzData"."85A1".I13 AND NOT "ST10_SysInput"."iE-StopPB"[1] AND NOT "ST10_SysInput"."iE-StopPB"[2] AND NOT "ST10_SysInput"."iE-StopPB"[3] AND NOT "ST10_SysInput"."iE-StopPB"[4] AND NOT "ST10_SysInput"."iE-StopPB"[5] AND NOT "ST10_SysInput"."iE-StopPB"[6] AND NOT "ST10_SysInput"."iE-StopPB"[7] AND NOT "ST10_SysInput"."iE-StopPB"[8] AND NOT "ST10_SysInput"."iE-StopPB"[9],
                           iResetFault := "ST10_SysInput".HMI_Button.ResetButton OR "Station_Sys".Alarm.Reset,
                           iModeSelectType := FALSE,
                           iManual := (("Station_Sys".Status.ModeSV = 1) AND "AlwaysFALSE") OR NOT "ST10_SysInput".HMI_Button."Manual/Auto",
                           iAuto := (("Station_Sys".Status.ModeSV = 2) AND "AlwaysFALSE") OR "ST10_SysInput".HMI_Button."Manual/Auto",
                           iHMIModeSelect := "Station_Sys".Status.ModeSV,
                           iControlOnMonitor := "ST10_SysInput".HMI_Button.ControlOn,
                           iSafetyDoor := 1,
                           iLightCurtain := true,
                           iMainPressureSwitch := "ST10_SysInput".Sys.iPressure,
                           iFixtureOK := true,
                           iChangeOverOK := "ST10_RecipeDB".Recipe.Equal OR "ChangeOver_DB".Global.ChangeOverSelected,
                           iInitializationOK := TRUE,
                           iAllDeviceOK := TRUE,
                           iAlarmOn := "Station_Sys".Alarm.ON,
                           iFlowRun := "Station_Sys".Auto.AllRun,
                           oReset => "Station_Sys".Cmd.Reset,
                           oEStopOK => "Station_Sys".Status.EStopOK,
                           oManualMode => "Station_Sys".Manual.Mode,
                           oAutoMode => "Station_Sys".Auto.Mode,
                           oOneCycleMode => "Station_Sys".Auto.OneCycleMode,
                           oStepMode => "Station_Sys".Auto.StepMode,
                           oRun => "Station_Sys".Status.Run,
                           "oEnable alarm" => "Station_Sys".Status.EnableAlarm,
                           oControlON => "Station_Sys".Status.ControlOn,
                           oMainPressureOK => "Station_Sys".Status.MainPressureOK,
                           oSafetyDoorOK => "Station_Sys".Safety.DoorOK[0],
                           oLightCurtainOK => "Station_Sys".Safety.LightCurtainOK[0],
                           oReady => "Station_Sys".Status.Ready,
                           oMode => "Station_Sys".Status.ModePV,
                           oStatus => "Station_Sys".Auto.Status);
   IF "AlwaysTRUE" AND NOT "ST10_SysInput".HMI_Button."Manual/Auto" THEN
       "Station_Sys".Status.ModeSV := 1;
   END_IF;
   IF "AlwaysTRUE" AND "ST10_SysInput".HMI_Button."Manual/Auto" THEN
       "Station_Sys".Status.ModeSV := 2;
   END_IF;
END_REGION

REGION Network 28: Start button
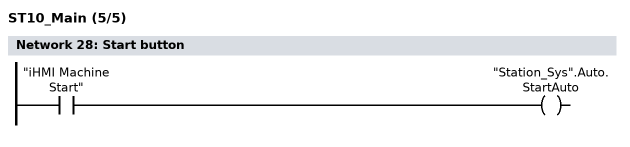
   RUNG wire#powerrail
      Contact( "iHMI Machine Start" )
      Coil( "Station_Sys".Auto.StartAuto )
   END_RUNG
   // the same network as SCL:
   "Station_Sys".Auto.StartAuto := "iHMI Machine Start";
END_REGION

REGION Network 29 (SCL): System Interface
   "Station_Sys".Interface.CPUFristCycle  := "Sys".COM.PLCRestarted;
   "Station_Sys".Interface.SysRun         := "Station_Sys".Status.Run;
   "Station_Sys".Interface.Reset          := "Station_Sys".Cmd.Reset;
   "Station_Sys".Interface.EstopOK        := "Station_Sys".Status.EStopOK;
   "Station_Sys".Interface.SafetyDoorOK   := "Station_Sys".Safety.DoorOK[0];
   "Station_Sys".Interface.LightCurtainOK := "Station_Sys".Safety.LightCurtainOK[0];
   "Station_Sys".Interface.SetInitial     := "Station_Sys".Initial.Set;
   "Station_Sys".Interface.InitialRun     := "Station_Sys".Initial.Running;
   "Station_Sys".Interface.Ready          := "Station_Sys".Status.Ready;
   "Station_Sys".Interface.ManualMode     := "Station_Sys".Manual.Mode;
   "Station_Sys".Interface.Auto           := "Station_Sys".Auto;
END_REGION

REGION Network 30: =====System Function related information Section =====End
END_REGION

REGION Network 31: CallCalibration//标定调用
END_REGION

REGION Network 32 (SCL): ByPass Button
   // A
   "ST10_GeneralData".FunctionDeSelect.A.FunctionDeSelected_Servo380A1  := "ST10_GeneralData".FunctionDeSelect.A.DeSelectPB_Servo380A1;
   "ST10_GeneralData".FunctionDeSelect.A.FunctionDeSelected_Servo381A1  := "ST10_GeneralData".FunctionDeSelect.A.DeSelectPB_Servo381A1;
   "ST10_GeneralData".FunctionDeSelect.A.FunctionDeSelected_Servo383A1  := "ST10_GeneralData".FunctionDeSelect.A.DeSelectPB_Servo383A1;
   "ST10_GeneralData".FunctionDeSelect.A.FunctionDeSelected_Reader800A1 := "ST10_GeneralData".FunctionDeSelect.A.DeSelectPB_Reader800A1;
   "ST10_GeneralData".FunctionDeSelect.A.FunctionDeSelected_Reader801A1 := "ST10_GeneralData".FunctionDeSelect.A.DeSelectPB_Reader801A1;
   "ST10_GeneralData".FunctionDeSelect.A.FunctionDeSelected_Reader802A1 := "ST10_GeneralData".FunctionDeSelect.A.DeSelectPB_Reader802A1;
   "ST10_GeneralData".FunctionDeSelect.A.FunctionDeSelected_Reader803A1 := "ST10_GeneralData".FunctionDeSelect.A.DeSelectPB_Reader803A1;
   "ST10_GeneralData".FunctionDeSelect.A.FunctionDeSelected_Reader804A1 := "ST10_GeneralData".FunctionDeSelect.A.DeSelectPB_Reader804A1;

   // B
   "ST10_GeneralData".FunctionDeSelect.B.FunctionDeSelected_Press372A1     := "ST10_GeneralData".FunctionDeSelect.B.DeSelectPB_Press372A1;
   "ST10_GeneralData".FunctionDeSelect.B.FunctionDeSelected_Press375A1     := "ST10_GeneralData".FunctionDeSelect.B.DeSelectPB_Press375A1;
   "ST10_GeneralData".FunctionDeSelect.B.FunctionDeSelected_Reader806A1    := "ST10_GeneralData".FunctionDeSelect.B.DeSelectPB_Reader806A1;
   "ST10_GeneralData".FunctionDeSelect.B.FunctionDeSelected_TestPress372A1 := "ST10_GeneralData".FunctionDeSelect.B.DeSelectPB_TestPress372A1;
   "ST10_GeneralData".FunctionDeSelect.B.FunctionDeSelected_TestPress375A1 := "ST10_GeneralData".FunctionDeSelect.B.DeSelectPB_TestPress375A1;

   // C
   "ST10_GeneralData".FunctionDeSelect.C.FunctionDeSelected_Servo382A1 := "ST10_GeneralData".FunctionDeSelect.C.DeSelectPB_Servo382A1;
   "ST10_GeneralData".FunctionDeSelect.C.FunctionDeSelected_ServoIAI := "ST10_GeneralData".FunctionDeSelect.C.DeSelectPB_ServoIAI;
   "ST10_GeneralData".FunctionDeSelect.C.FunctionDeSelected_IV3810A1 := "ST10_GeneralData".FunctionDeSelect.C.DeSelectPB_IV3810A1;
   "ST10_GeneralData".FunctionDeSelect.C.FunctionDeSelected_IV3811A1 := "ST10_GeneralData".FunctionDeSelect.C.DeSelectPB_IV3811A1;
   "ST10_GeneralData".FunctionDeSelect.C.FunctionDeSelected_Glue := "ST10_GeneralData".FunctionDeSelect.C.DeSelectPB_Glue;

   // E
   "ST10_GeneralData".FunctionDeSelect.E.FunctionDeSelected := "ST10_GeneralData".FunctionDeSelect.E.DeSelectPB;

   // F
   "ST10_GeneralData".FunctionDeSelect.F.FunctionDeSelected_Reader805A1 := "ST10_GeneralData".FunctionDeSelect.F.DeSelectPB_Reader805A1;

   // H
   "ST10_GeneralData".FunctionDeSelect.H.FunctionDeSelected := "ST10_GeneralData".FunctionDeSelect.H.DeSelectPB;

   // J
   "ST10_GeneralData".FunctionDeSelect.J.FunctionDeSelected := "ST10_GeneralData".FunctionDeSelect.J.DeSelectPB;

   // K
   "ST10_GeneralData".FunctionDeSelect.K.FunctionDeSelected := "ST10_GeneralData".FunctionDeSelect.K.DeSelectPB;

   // L
   "ST10_GeneralData".FunctionDeSelect.L.FunctionDeSelected := "ST10_GeneralData".FunctionDeSelect.L.DeSelectPB;

   // MES
   "ST10_GeneralData".FunctionDeSelect.MES.FunctionDeSelected := "ST10_GeneralData".FunctionDeSelect.MES.DeSelectPB;

   //Auto>Maanual  ScanFixture
   "ST10_GeneralData".FunctionDeSelect.Global.FunctionDeSelected_ScanFixture := "ST10_GeneralData".FunctionDeSelect.Global.DeSelectPB_ScanFixture;
END_REGION
END_FUNCTION

FUNCTION "ST10_Input" : Void   // FC1001, LAD
{ S7_Optimized_Access := 'FALSE' }
// 注：本程序用来处理需要滤波，延时、计算的输入信号
// stored: AutoNumber false, SetENOAutomatically false
BEGIN

REGION Network 1 (SCL): HMI信号映射 / HMI signal mapping
   "ST10_SysInput".HMI_Button.ControlOn := "iHMI Control On";
   //"ST350_SysInput".HMI_Button.ControlOff:=
   "ST10_SysInput".HMI_Button.MachineStart := "iHMI Machine Start";
   "ST10_SysInput".HMI_Button.MachineStop := "iHMI Machine Stop";
   "ST10_SysInput".HMI_Button.ResetButton := "iHMI ResetButton";
   "ST10_SysInput".HMI_Button."Manual/Auto" := "iHMI Manual/Auto";
   "ST10_SysInput".HMI_Button.SafetyGateUnlock := "iHMI Safety Gate Unlock";
   "ST10_SysInput".HMI_Button."E-Stop" :=  "iHMI E-Stop";
END_REGION

REGION Network 2 (SCL): Sys IO Image
   "ST10_SysInput".Sys.iCircuitBreakerOK1 := "iCircuit Breaker OK_1";
   "ST10_SysInput".Sys.iCircuitBreakerOK2 := "iCircuit Breaker OK_2";
   "ST10_SysInput".Sys.iPressure:= "iPressure";
END_REGION

REGION Network 3 (SCL): iE-StopPB
   "ST10_SysInput"."iE-StopPB"[1] := "iE_StopButton2_A01";
   "ST10_SysInput"."iE-StopPB"[2] := "iE_StopButton3_A02";
   "ST10_SysInput"."iE-StopPB"[3] := "iE_StopButton4_H";
   "ST10_SysInput"."iE-StopPB"[4] := "iE_StopButton5_J";
   "ST10_SysInput"."iE-StopPB"[5] := "iE_StopButton6_K";
   "ST10_SysInput"."iE-StopPB"[6] := "iE_StopButton7_L";
   "ST10_SysInput"."iE-StopPB"[7] := "iH_StopButton";
   "ST10_SysInput"."iE-StopPB"[8] := "iJ_StopButton";
   "ST10_SysInput"."iE-StopPB"[9] := "iK_StopButton";
END_REGION

REGION Network 4 (SCL): iSafetyGatFeedBack
   (*
   "ST350_SysInput".iSafetyGatFeedBack[1] := "iSafety door Locking FeedBack_1";
   "ST350_SysInput".iSafetyGatFeedBack[2] := "iSafety door Locking FeedBack_2";
   "ST350_SysInput".iSafetyGatFeedBack[3] := "iSafety door Locking FeedBack_3";
   "ST350_SysInput".iSafetyGatFeedBack[4] := "iSafety door Locking FeedBack_4";
   "ST350_SysInput".iSafetyGatFeedBack[5] := "iSafety door Locking FeedBack_5";
   "ST350_SysInput".iSafetyGatFeedBack[6] := "iSafety door Locking FeedBack_6";
   "ST350_SysInput".iSafetyGatFeedBack[7] := "iSafety door Locking FeedBack_7";
   "ST350_SysInput".iSafetyGatFeedBack[8] := "iSafety door Locking FeedBack_8";
   *)
END_REGION

REGION Network 5 (SCL): iSafetydoorLockingFeedBack
   "ST10_SysInput".iSafetydoorLockingFeedBack[1] := "iSafety door Locking FeedBack_1";
   "ST10_SysInput".iSafetydoorLockingFeedBack[2] := "iSafety door Locking FeedBack_2";
   "ST10_SysInput".iSafetydoorLockingFeedBack[3] := "iSafety door Locking FeedBack_3";
   "ST10_SysInput".iSafetydoorLockingFeedBack[4] := "iSafety door Locking FeedBack_4";
   "ST10_SysInput".iSafetydoorLockingFeedBack[5] := "iSafety door Locking FeedBack_5";
   "ST10_SysInput".iSafetydoorLockingFeedBack[6] := "iSafety door Locking FeedBack_6";
   "ST10_SysInput".iSafetydoorLockingFeedBack[7] := "iSafety door Locking FeedBack_7";
   "ST10_SysInput".iSafetydoorLockingFeedBack[8] := "iSafety door Locking FeedBack_8";
END_REGION

REGION Network 6 (SCL): iSafetydoorLockingFeedBack
   "ST10_SysInput".iMaterieldoorLockingFeedBack[1] := "iMateriel Door Locking FeedBack_H1";
   "ST10_SysInput".iMaterieldoorLockingFeedBack[2] := "iMateriel Door Locking FeedBack_H2";
   "ST10_SysInput".iMaterieldoorLockingFeedBack[3] := "iMateriel Door Locking FeedBack_J1";
   "ST10_SysInput".iMaterieldoorLockingFeedBack[4] := "iMateriel Door Locking FeedBack_J2";
   "ST10_SysInput".iMaterieldoorLockingFeedBack[5] := "iMateriel Door Locking FeedBack_K1";
   "ST10_SysInput".iMaterieldoorLockingFeedBack[6] := "iMateriel Door Locking FeedBack_K2";
   "ST10_SysInput".iMaterieldoorLockingFeedBack[7] := "iMateriel Door Locking FeedBack_L1";
END_REGION
END_FUNCTION

FUNCTION "ST10_Alarm" : Void   // FC1005, LAD
{ S7_Optimized_Access := 'FALSE' }
// stored: AutoNumber false, SetENOAutomatically false
   VAR_TEMP
      tpAlarm : Array[0..2, 0..15] of Bool;
      tpAlarmInt AT tpAlarm : Array[0..2] of Int;
      tpTP : Array[0..1] of Int;
      tpClear : Byte;
      FixtureNumber : Int;
      i : Int;
      tpAlwayoff : Bool;
   END_VAR
   VAR_TEMP   // added for the SCL form of the ladder/FBD networks
      _w1 : Bool;
      _w2 : Bool;
      _w3 : Bool;
   END_VAR
BEGIN

REGION Network 1: Normal off
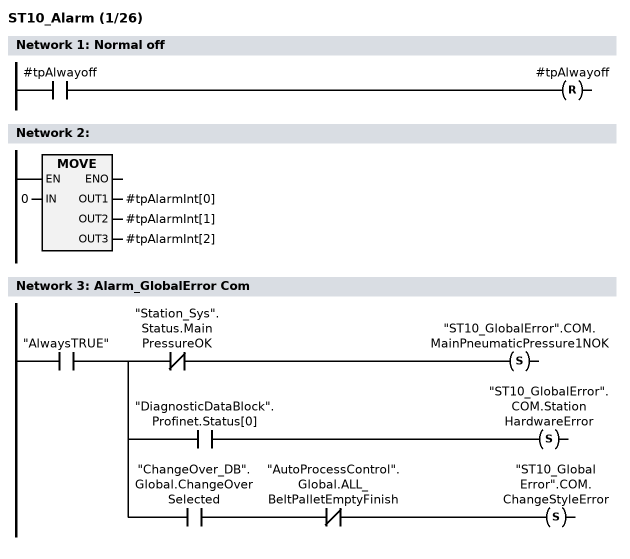
   RUNG wire#powerrail
      Contact( #tpAlwayoff )
      R_Coil( #tpAlwayoff )
   END_RUNG
   // the same network as SCL:
   IF #tpAlwayoff THEN #tpAlwayoff := FALSE; END_IF;
END_REGION

REGION Network 2
   RUNG wire#powerrail
      Move(in := 0, out1 => #tpAlarmInt[0], out2 => #tpAlarmInt[1], out3 => #tpAlarmInt[2])
   END_RUNG
   // the same network as SCL:
   #tpAlarmInt[0] := 0;
   #tpAlarmInt[1] := 0;
   #tpAlarmInt[2] := 0;
END_REGION

REGION Network 3: Alarm_GlobalError Com
   RUNG wire#powerrail
      Contact( "AlwaysTRUE" )
      wire#w1
      I_Contact( "Station_Sys".Status.MainPressureOK )
      S_Coil( "ST10_GlobalError".COM.MainPneumaticPressure1NOK )
   END_RUNG
   RUNG wire#w1
      Contact( "DiagnosticDataBlock".Profinet.Status[0] )
      S_Coil( "ST10_GlobalError".COM.StationHardwareError )
   END_RUNG
   RUNG wire#w1
      Contact( "ChangeOver_DB".Global.ChangeOverSelected )
      I_Contact( "AutoProcessControl".Global.ALL_BeltPalletEmptyFinish )
      S_Coil( "ST10_GlobalError".COM.ChangeStyleError )
   END_RUNG
   // the same network as SCL:
   IF "AlwaysTRUE" AND NOT "Station_Sys".Status.MainPressureOK THEN
       "ST10_GlobalError".COM.MainPneumaticPressure1NOK := TRUE;
   END_IF;
   IF "AlwaysTRUE" AND "DiagnosticDataBlock".Profinet.Status[0] THEN
       "ST10_GlobalError".COM.StationHardwareError := TRUE;
   END_IF;
   IF "AlwaysTRUE" AND "ChangeOver_DB".Global.ChangeOverSelected AND NOT "AutoProcessControl".Global.ALL_BeltPalletEmptyFinish THEN
       "ST10_GlobalError".COM.ChangeStyleError := TRUE;
   END_IF;
END_REGION

